SPLINE
SPL {X  -162.820, Y  +495.897, Z    +0.000, E1   +21.662, E3 +486078.194}
SPL {X  -162.820, Y  +493.717, Z    +0.000, E1   +21.704, E3 +486089.301}
SPL {X  -162.820, Y  +491.396, Z    +0.000, E1   +21.707, E3 +486101.424}
SPL {X  -162.820, Y  +489.485, Z    +0.000, E1   +21.661, E3 +486111.772}
SPL {X  -162.820, Y  +487.723, Z    +0.000, E1   +21.665, E3 +486120.976}
SPL {X  -162.820, Y  +485.661, Z    +0.000, E1   +21.712, E3 +486131.419}
SPL {X  -162.820, Y  +482.775, Z    +0.000, E1   +21.716, E3 +486146.672}
SPL {X  -162.820, Y  +479.894, Z    +0.000, E1   +21.695, E3 +486161.748}
SPL {X  -162.820, Y  +477.685, Z    +0.000, E1   +21.656, E3 +486173.685}
SPL {X  -162.820, Y  +475.419, Z    +0.000, E1   +21.711, E3 +486185.038}
SPL {X  -162.820, Y  +473.301, Z    +0.000, E1   +21.712, E3 +486196.135}
SPL {X  -162.820, Y  +470.965, Z    +0.000, E1   +21.700, E3 +486208.480}
SPL {X  -162.820, Y  +469.036, Z    +0.000, E1   +21.695, E3 +486218.524}
SPL {X  -162.820, Y  +467.138, Z    +0.000, E1   +21.678, E3 +486228.695}
SPL {X  -162.820, Y  +465.011, Z    +0.000, E1   +21.692, E3 +486239.678}
SPL {X  -162.820, Y  +462.669, Z    +0.000, E1   +21.752, E3 +486251.459}
SPL {X  -162.820, Y  +460.725, Z    +0.000, E1   +21.689, E3 +486262.072}
SPL {X  -162.820, Y  +458.666, Z    +0.000, E1   +21.695, E3 +486272.883}
SPL {X  -162.820, Y  +456.431, Z    +0.000, E1   +21.708, E3 +486284.412}
SPL {X  -162.820, Y  +453.609, Z    +0.000, E1   +21.757, E3 +486298.946}
SPL {X  -162.820, Y  +450.610, Z    +0.000, E1   +21.698, E3 +486315.003}
SPL {X  -162.820, Y  +448.170, Z    +0.000, E1   +21.667, E3 +486328.024}
SPL {X  -162.820, Y  +446.246, Z    +0.000, E1   +21.696, E3 +486337.842}
SPL {X  -162.820, Y  +443.784, Z    +0.000, E1   +21.713, E3 +486350.628}
SPL {X  -162.820, Y  +441.754, Z    +0.000, E1   +21.708, E3 +486361.180}
SPL {X  -162.820, Y  +439.933, Z    +0.000, E1   +21.690, E3 +486370.944}
SPL {X  -162.820, Y  +437.628, Z    +0.000, E1   +21.678, E3 +486383.132}
SPL {X  -162.820, Y  +435.262, Z    +0.000, E1   +21.727, E3 +486395.067}
SPL {X  -162.820, Y  +433.510, Z    +0.000, E1   +21.692, E3 +486404.481}
SPL {X  -162.820, Y  +431.492, Z    +0.000, E1   +21.686, E3 +486415.177}
SPL {X  -162.820, Y  +429.074, Z    +0.000, E1   +21.710, E3 +486427.629}
SPL {X  -162.820, Y  +427.020, Z    +0.000, E1   +21.674, E3 +486438.630}
SPL {X  -162.820, Y  +424.525, Z    +0.000, E1   +21.712, E3 +486451.543}
SPL {X  -162.820, Y  +421.144, Z    +0.000, E1   +21.719, E3 +486469.210}
SPL {X  -162.820, Y  +418.116, Z    +0.000, E1   +21.761, E3 +486484.541}
SPL {X  -162.820, Y  +416.127, Z    +0.000, E1   +21.715, E3 +486495.247}
SPL {X  -162.820, Y  +414.361, Z    +0.000, E1   +21.613, E3 +486505.434}
SPL {X  -162.820, Y  +412.134, Z    +0.000, E1   +21.697, E3 +486516.378}
SPL {X  -162.820, Y  +409.248, Z    +0.000, E1   +21.741, E3 +486531.314}
SPL {X  -162.820, Y  +406.238, Z    +0.000, E1   +21.697, E3 +486547.282}
SPL {X  -162.820, Y  +404.001, Z    +0.000, E1   +21.723, E3 +486558.711}
SPL {X  -162.820, Y  +402.223, Z    +0.000, E1   +21.697, E3 +486568.196}
SPL {X  -162.820, Y  +400.348, Z    +0.000, E1   +21.713, E3 +486577.922}
SPL {X  -162.820, Y  +398.298, Z    +0.000, E1   +21.721, E3 +486588.538}
SPL {X  -162.820, Y  +396.371, Z    +0.000, E1   +21.713, E3 +486598.720}
SPL {X  -162.820, Y  +394.508, Z    +0.000, E1   +21.616, E3 +486609.275}
SPL {X  -162.820, Y  +392.435, Z    +0.000, E1   +21.681, E3 +486619.629}
SPL {X  -162.820, Y  +389.390, Z    +0.000, E1   +21.742, E3 +486635.235}
SPL {X  -162.820, Y  +386.818, Z    +0.000, E1   +21.679, E3 +486648.994}
SPL {X  -162.820, Y  +384.697, Z    +0.000, E1   +21.693, E3 +486660.064}
SPL {X  -162.820, Y  +382.288, Z    +0.000, E1   +21.742, E3 +486672.188}
SPL {X  -162.817, Y  +379.520, Z    +0.000, E1   +21.723, E3 +486687.025}
SPL {X  -162.776, Y  +376.710, Z    +0.000, E1   +21.698, E3 +486701.765}
SPL {X  -162.707, Y  +374.438, Z    +0.000, E1   +21.688, E3 +486713.768}
SPL {X  -162.607, Y  +372.171, Z    +0.000, E1   +21.692, E3 +486725.568}
SPL {X  -162.494, Y  +370.197, Z    +0.000, E1   +21.655, E3 +486736.194}
SPL {X  -162.349, Y  +368.131, Z    +0.000, E1   +21.624, E3 +486747.312}
SPL {X  -162.161, Y  +365.866, Z    +0.000, E1   +21.642, E3 +486758.998}
SPL {X  -161.651, Y  +361.024, Z    +0.000, E1   +22.970, E3 +486772.421}
SPL {X  -160.281, Y  +351.857, Z    +0.000, E1   +24.243, E3 +486807.760}
ENDSPLINE

SPLINE
SPL {X  -161.833, Y  +362.603, Z    +0.000, E1   +17.021, E3 +486822.456}
ENDSPLINE

SPLINE
SPL {X  -160.786, Y  +354.842, Z    +0.000, E1   +19.274, E3 +486854.611}
ENDSPLINE

SPLINE
SPL {X  -162.485, Y  +370.062, Z    +0.000, E1   +10.606, E3 +486860.990}
SPL {X  -162.818, Y  +379.636, Z    +0.000, E1    +5.115, E3 +486850.338}
SPL {X  -162.820, Y  +386.976, Z    +0.000, E1    +0.144, E3 +486849.437}
SPL {X  -162.820, Y  +391.982, Z    +0.000, E1    -3.443, E3 +486856.202}
SPL {X  -162.820, Y  +399.630, Z    +0.000, E1    -9.426, E3 +486858.710}
SPL {X  -162.820, Y  +408.127, Z    +0.000, E1   -18.417, E3 +486844.998}
SPL {X  -162.820, Y  +420.083, Z    +0.000, E1   -24.325, E3 +486865.474}
SPL {X  -162.820, Y  +428.527, Z    +0.000, E1   -26.988, E3 +486882.766}
SPL {X  -162.820, Y  +431.336, Z    +0.000, E1   -24.162, E3 +486912.976}
SPL {X  -162.820, Y  +432.048, Z    +0.000, E1   -22.832, E3 +486927.480}
SPL {X  -162.820, Y  +434.888, Z    +0.000, E1   -22.823, E3 +486941.429}
SPL {X  -162.820, Y  +436.834, Z    +0.000, E1   -22.779, E3 +486951.389}
SPL {X  -162.820, Y  +438.868, Z    +0.000, E1   -22.837, E3 +486961.043}
SPL {X  -162.820, Y  +441.351, Z    +0.000, E1   -22.805, E3 +486973.618}
SPL {X  -162.820, Y  +443.809, Z    +0.000, E1   -22.804, E3 +486985.784}
SPL {X  -162.820, Y  +447.077, Z    +0.000, E1   -22.869, E3 +487001.595}
SPL {X  -162.820, Y  +449.911, Z    +0.000, E1   -22.774, E3 +487016.204}
SPL {X  -162.820, Y  +451.861, Z    +0.000, E1   -22.750, E3 +487026.052}
SPL {X  -162.820, Y  +454.167, Z    +0.000, E1   -22.842, E3 +487036.781}
SPL {X  -162.820, Y  +456.529, Z    +0.000, E1   -22.855, E3 +487048.310}
SPL {X  -162.820, Y  +458.725, Z    +0.000, E1   -22.793, E3 +487059.714}
SPL {X  -162.820, Y  +461.700, Z    +0.000, E1   -22.822, E3 +487074.336}
SPL {X  -162.820, Y  +464.633, Z    +0.000, E1   -22.813, E3 +487088.833}
SPL {X  -162.820, Y  +466.699, Z    +0.000, E1   -22.824, E3 +487098.879}
SPL {X  -162.820, Y  +468.655, Z    +0.000, E1   -22.858, E3 +487108.323}
SPL {X  -162.820, Y  +470.892, Z    +0.000, E1   -22.837, E3 +487119.562}
SPL {X  -162.820, Y  +473.485, Z    +0.000, E1   -22.806, E3 +487132.760}
SPL {X  -162.820, Y  +475.738, Z    +0.000, E1   -22.728, E3 +487144.425}
SPL {X  -162.820, Y  +478.177, Z    +0.000, E1   -22.834, E3 +487155.765}
SPL {X  -162.820, Y  +481.034, Z    +0.000, E1   -22.831, E3 +487169.902}
SPL {X  -162.820, Y  +483.391, Z    +0.000, E1   -22.793, E3 +487181.838}
SPL {X  -162.820, Y  +486.307, Z    +0.000, E1   -22.833, E3 +487196.092}
SPL {X  -162.820, Y  +489.750, Z    +0.000, E1   -22.832, E3 +487213.162}
SPL {X  -162.820, Y  +492.546, Z    +0.000, E1   -22.823, E3 +487226.920}
SPL {X  -162.820, Y  +495.526, Z    +0.000, E1   -22.833, E3 +487241.803}
SPL {X  -162.820, Y  +499.330, Z    +0.000, E1   -22.841, E3 +487260.584}
SPL {X  -162.820, Y  +502.361, Z    +0.000, E1   -22.801, E3 +487275.743}
SPL {X  -162.820, Y  +505.323, Z    +0.000, E1   -22.838, E3 +487290.215}
SPL {X  -162.820, Y  +508.611, Z    +0.000, E1   -22.838, E3 +487306.477}
SPL {X  -162.820, Y  +511.620, Z    +0.000, E1   -22.791, E3 +487321.721}
SPL {X  -162.820, Y  +513.873, Z    +0.000, E1   -22.800, E3 +487332.693}
SPL {X  -162.820, Y  +516.100, Z    +0.000, E1   -22.809, E3 +487343.770}
SPL {X  -162.820, Y  +518.662, Z    +0.000, E1   -22.847, E3 +487356.068}
SPL {X  -162.820, Y  +520.641, Z    +0.000, E1   -22.790, E3 +487366.309}
SPL {X  -162.820, Y  +522.740, Z    +0.000, E1   -22.811, E3 +487376.552}
SPL {X  -162.820, Y  +524.628, Z    +0.000, E1   -22.846, E3 +487385.547}
SPL {X  -162.820, Y  +526.661, Z    +0.000, E1   -22.801, E3 +487396.102}
SPL {X  -162.820, Y  +529.662, Z    +0.000, E1   -22.810, E3 +487410.953}
SPL {X  -162.820, Y  +532.614, Z    +0.000, E1   -22.828, E3 +487425.359}
SPL {X  -162.820, Y  +534.838, Z    +0.000, E1   -22.864, E3 +487435.988}
SPL {X  -162.820, Y  +536.882, Z    +0.000, E1   -22.782, E3 +487446.843}
SPL {X  -162.820, Y  +539.194, Z    +0.000, E1   -22.826, E3 +487457.891}
SPL {X  -162.820, Y  +541.555, Z    +0.000, E1   -22.817, E3 +487469.706}
SPL {X  -162.820, Y  +543.728, Z    +0.000, E1   -22.799, E3 +487480.563}
SPL {X  -162.820, Y  +545.925, Z    +0.000, E1   -22.803, E3 +487491.433}
SPL {X  -162.820, Y  +548.328, Z    +0.000, E1   -22.796, E3 +487503.429}
SPL {X  -162.820, Y  +551.027, Z    +0.000, E1   -22.819, E3 +487516.622}
SPL {X  -162.820, Y  +553.721, Z    +0.000, E1   -22.807, E3 +487530.066}
SPL {X  -162.820, Y  +556.430, Z    +0.000, E1   -22.821, E3 +487543.362}
SPL {X  -162.820, Y  +559.675, Z    +0.000, E1   -22.837, E3 +487559.442}
SPL {X  -162.820, Y  +562.799, Z    +0.000, E1   -22.814, E3 +487574.948}
SPL {X  -162.820, Y  +565.170, Z    +0.000, E1   -22.801, E3 +487586.773}
SPL {X  -162.820, Y  +568.020, Z    +0.000, E1   -22.787, E3 +487601.160}
SPL {X  -162.820, Y  +570.992, Z    +0.000, E1   -22.834, E3 +487615.379}
SPL {X  -162.820, Y  +572.901, Z    +0.000, E1   -22.775, E3 +487625.247}
SPL {X  -162.820, Y  +575.638, Z    +0.000, E1   -22.855, E3 +487638.357}
SPL {X  -162.820, Y  +578.553, Z    +0.000, E1   -22.801, E3 +487653.069}
SPL {X  -162.820, Y  +581.064, Z    +0.000, E1   -22.823, E3 +487665.354}
SPL {X  -162.820, Y  +583.435, Z    +0.000, E1   -22.808, E3 +487677.175}
SPL {X  -162.820, Y  +585.410, Z    +0.000, E1   -22.764, E3 +487687.311}
SPL {X  -162.820, Y  +587.676, Z    +0.000, E1   -22.853, E3 +487697.826}
SPL {X  -162.820, Y  +589.682, Z    +0.000, E1   -22.776, E3 +487708.355}
SPL {X  -162.820, Y  +591.720, Z    +0.000, E1   -22.868, E3 +487717.666}
SPL {X  -162.820, Y  +593.650, Z    +0.000, E1   -22.810, E3 +487727.736}
SPL {X  -162.820, Y  +595.830, Z    +0.000, E1   -22.828, E3 +487738.352}
SPL {X  -162.820, Y  +598.094, Z    +0.000, E1   -22.843, E3 +487749.465}
SPL {X  -162.820, Y  +600.420, Z    +0.000, E1   -22.826, E3 +487761.096}
SPL {X  -162.820, Y  +602.573, Z    +0.000, E1   -22.830, E3 +487771.682}
SPL {X  -162.820, Y  +604.828, Z    +0.000, E1   -22.784, E3 +487783.320}
SPL {X  -162.820, Y  +607.142, Z    +0.000, E1   -22.808, E3 +487794.501}
SPL {X  -162.820, Y  +608.890, Z    +0.000, E1   -22.790, E3 +487803.325}
SPL {X  -162.820, Y  +611.103, Z    +0.000, E1   -22.785, E3 +487814.363}
SPL {X  -162.820, Y  +613.294, Z    +0.000, E1   -22.780, E3 +487825.237}
SPL {X  -162.820, Y  +615.356, Z    +0.000, E1   -22.799, E3 +487835.294}
SPL {X  -162.820, Y  +617.439, Z    +0.000, E1   -22.808, E3 +487845.552}
SPL {X  -162.820, Y  +619.665, Z    +0.000, E1   -22.817, E3 +487856.520}
SPL {X  -162.820, Y  +621.733, Z    +0.000, E1   -22.759, E3 +487867.244}
SPL {X  -162.820, Y  +624.076, Z    +0.000, E1   -22.774, E3 +487878.749}
SPL {X  -162.820, Y  +626.527, Z    +0.000, E1   -22.768, E3 +487890.992}
SPL {X  -162.820, Y  +629.758, Z    +0.000, E1   -22.800, E3 +487906.921}
SPL {X  -162.820, Y  +632.572, Z    +0.000, E1   -22.785, E3 +487920.770}
SPL {X  -162.820, Y  +634.507, Z    +0.000, E1   -22.784, E3 +487930.409}
SPL {X  -162.820, Y  +636.863, Z    +0.000, E1   -22.760, E3 +487942.331}
SPL {X  -162.820, Y  +640.111, Z    +0.000, E1   -22.809, E3 +487958.214}
SPL {X  -162.820, Y  +643.449, Z    +0.000, E1   -22.796, E3 +487974.731}
SPL {X  -162.820, Y  +645.630, Z    +0.000, E1   -22.795, E3 +487985.428}
SPL {X  -162.820, Y  +647.561, Z    +0.000, E1   -22.705, E3 +487995.878}
SPL {X  -162.820, Y  +649.758, Z    +0.000, E1   -22.780, E3 +488006.068}
SPL {X  -162.820, Y  +651.708, Z    +0.000, E1   -22.810, E3 +488015.563}
SPL {X  -162.820, Y  +653.898, Z    +0.000, E1   -22.796, E3 +488026.484}
SPL {X  -162.820, Y  +656.161, Z    +0.000, E1   -22.812, E3 +488037.605}
SPL {X  -162.820, Y  +658.384, Z    +0.000, E1   -22.822, E3 +488048.471}
SPL {X  -162.820, Y  +660.215, Z    +0.000, E1   -22.649, E3 +488059.062}
SPL {X  -162.820, Y  +662.823, Z    +0.000, E1   -22.799, E3 +488070.770}
SPL {X  -162.820, Y  +665.112, Z    +0.000, E1   -22.835, E3 +488081.824}
SPL {X  -162.820, Y  +667.016, Z    +0.000, E1   -22.823, E3 +488091.253}
SPL {X  -162.820, Y  +668.960, Z    +0.000, E1   -22.773, E3 +488101.420}
SPL {X  -162.820, Y  +672.333, Z    +0.000, E1   -22.837, E3 +488117.756}
SPL {X  -162.812, Y  +675.071, Z    +0.000, E1   -22.742, E3 +488131.901}
SPL {X  -162.773, Y  +677.428, Z    +0.000, E1   -22.762, E3 +488143.499}
SPL {X  -162.691, Y  +679.987, Z    +0.000, E1   -22.794, E3 +488155.912}
SPL {X  -162.604, Y  +681.880, Z    +0.000, E1   -22.691, E3 +488166.073}
SPL {X  -162.458, Y  +684.346, Z    +0.000, E1   -22.764, E3 +488177.866}
SPL {X  -162.296, Y  +686.547, Z    +0.000, E1   -22.660, E3 +488189.483}
SPL {X  -162.090, Y  +688.902, Z    +0.000, E1   -22.700, E3 +488200.991}
SPL {X  -161.474, Y  +694.390, Z    +0.000, E1   -24.298, E3 +488214.347}
SPL {X  -158.730, Y  +709.763, Z    +0.000, E1   -31.225, E3 +488225.685}
ENDSPLINE

SPLINE
SPL {X  -160.932, Y  +698.225, Z    +0.000, E1   -21.712, E3 +488256.795}
SPL {X  -161.917, Y  +690.622, Z    +0.000, E1   -16.445, E3 +488270.395}
ENDSPLINE

SPLINE
SPL {X  -161.349, Y  +695.340, Z    +0.000, E1   -18.625, E3 +488278.014}
ENDSPLINE

SPLINE
SPL {X  -162.534, Y  +683.153, Z    +0.000, E1   -10.475, E3 +488299.144}
SPL {X  -162.820, Y  +667.630, Z    +0.000, E1    -0.882, E3 +488293.121}
SPL {X  -162.820, Y  +661.883, Z    +0.000, E1    +3.373, E3 +488298.564}
SPL {X  -162.820, Y  +653.808, Z    +0.000, E1    +9.891, E3 +488296.255}
SPL {X  -162.820, Y  +632.548, Z    +0.000, E1   +27.446, E3 +488292.792}
ENDSPLINE

SPLINE
SPL {X  -162.820, Y  +638.080, Z    +0.000, E1   +18.858, E3 +488320.540}
ENDSPLINE

SPLINE
SPL {X  -162.820, Y  +623.278, Z    +0.000, E1   +28.723, E3 +488322.111}
SPL {X  -162.820, Y  +618.658, Z    +0.000, E1   +26.841, E3 +488350.720}
ENDSPLINE

SPLINE
SPL {X  -162.820, Y  +623.685, Z    +0.000, E1   +22.346, E3 +488363.027}
ENDSPLINE

SPLINE
SPL {X  -162.820, Y  +621.304, Z    +0.000, E1   +22.259, E3 +488375.842}
SPL {X  -162.820, Y  +618.758, Z    +0.000, E1   +22.239, E3 +488388.993}
SPL {X  -162.820, Y  +616.062, Z    +0.000, E1   +22.275, E3 +488402.413}
SPL {X  -162.820, Y  +613.536, Z    +0.000, E1   +22.242, E3 +488415.535}
SPL {X  -162.820, Y  +610.461, Z    +0.000, E1   +22.264, E3 +488431.166}
SPL {X  -162.820, Y  +607.796, Z    +0.000, E1   +22.261, E3 +488444.537}
SPL {X  -162.820, Y  +605.178, Z    +0.000, E1   +22.267, E3 +488458.021}
SPL {X  -162.820, Y  +602.350, Z    +0.000, E1   +22.224, E3 +488472.638}
SPL {X  -162.820, Y  +599.842, Z    +0.000, E1   +22.298, E3 +488484.790}
SPL {X  -162.820, Y  +597.194, Z    +0.000, E1   +22.253, E3 +488498.711}
SPL {X  -162.820, Y  +594.779, Z    +0.000, E1   +22.284, E3 +488510.615}
SPL {X  -162.820, Y  +592.389, Z    +0.000, E1   +22.245, E3 +488523.231}
SPL {X  -162.820, Y  +589.492, Z    +0.000, E1   +22.304, E3 +488537.415}
SPL {X  -162.820, Y  +587.447, Z    +0.000, E1   +22.279, E3 +488547.944}
SPL {X  -162.820, Y  +585.192, Z    +0.000, E1   +22.298, E3 +488559.355}
SPL {X  -162.820, Y  +582.610, Z    +0.000, E1   +22.234, E3 +488572.978}
SPL {X  -162.820, Y  +580.317, Z    +0.000, E1   +22.300, E3 +488584.032}
SPL {X  -162.820, Y  +578.878, Z    +0.000, E1   +22.272, E3 +488591.541}
SPL {X  -162.820, Y  +576.856, Z    +0.000, E1   +22.233, E3 +488602.300}
SPL {X  -162.820, Y  +574.811, Z    +0.000, E1   +22.236, E3 +488612.563}
SPL {X  -162.820, Y  +572.645, Z    +0.000, E1   +22.246, E3 +488623.659}
SPL {X  -162.820, Y  +570.282, Z    +0.000, E1   +22.231, E3 +488635.709}
SPL {X  -162.820, Y  +567.961, Z    +0.000, E1   +22.247, E3 +488647.499}
SPL {X  -162.820, Y  +564.506, Z    +0.000, E1   +22.298, E3 +488664.813}
SPL {X  -162.820, Y  +561.620, Z    +0.000, E1   +22.191, E3 +488680.194}
SPL {X  -162.820, Y  +559.515, Z    +0.000, E1   +22.273, E3 +488690.196}
SPL {X  -162.820, Y  +556.723, Z    +0.000, E1   +22.309, E3 +488704.279}
SPL {X  -162.820, Y  +554.378, Z    +0.000, E1   +22.288, E3 +488716.125}
SPL {X  -162.820, Y  +552.787, Z    +0.000, E1   +22.213, E3 +488724.947}
SPL {X  -162.820, Y  +550.871, Z    +0.000, E1   +22.229, E3 +488734.541}
SPL {X  -162.820, Y  +548.168, Z    +0.000, E1   +22.298, E3 +488747.877}
SPL {X  -162.820, Y  +545.860, Z    +0.000, E1   +22.216, E3 +488760.135}
SPL {X  -162.820, Y  +543.558, Z    +0.000, E1   +22.285, E3 +488771.365}
SPL {X  -162.820, Y  +541.633, Z    +0.000, E1   +22.257, E3 +488781.294}
SPL {X  -162.820, Y  +539.116, Z    +0.000, E1   +22.302, E3 +488793.904}
SPL {X  -162.820, Y  +535.523, Z    +0.000, E1   +22.266, E3 +488812.566}
SPL {X  -162.820, Y  +531.757, Z    +0.000, E1   +22.276, E3 +488831.620}
SPL {X  -162.820, Y  +527.980, Z    +0.000, E1   +22.326, E3 +488850.451}
SPL {X  -162.820, Y  +524.599, Z    +0.000, E1   +22.287, E3 +488867.849}
SPL {X  -162.820, Y  +522.011, Z    +0.000, E1   +22.282, E3 +488880.926}
SPL {X  -162.820, Y  +519.457, Z    +0.000, E1   +22.481, E3 +488892.215}
SPL {X  -162.820, Y  +506.285, Z    +0.000, E1   +28.538, E3 +488903.673}
SPL {X  -162.820, Y  +504.441, Z    +0.000, E1   +27.574, E3 +488918.015}
SPL {X  -162.820, Y  +502.813, Z    +0.000, E1   +26.013, E3 +488936.213}
SPL {X  -162.820, Y  +502.016, Z    +0.000, E1   +24.802, E3 +488948.555}
SPL {X  -162.820, Y  +501.060, Z    +0.000, E1   +24.081, E3 +488958.745}
SPL {X  -162.820, Y  +500.336, Z    +0.000, E1   +23.110, E3 +488969.885}
SPL {X  -162.820, Y  +499.240, Z    +0.000, E1   +22.316, E3 +488982.196}
SPL {X  -162.820, Y  +498.027, Z    +0.000, E1   +21.516, E3 +488995.103}
SPL {X  -162.820, Y  +495.897, Z    +0.000, E1   +21.662, E3 +489005.023}
SPL {X  -162.820, Y  +493.717, Z    +0.000, E1   +21.704, E3 +489016.130}
SPL {X  -162.820, Y  +491.396, Z    +0.000, E1   +21.707, E3 +489028.254}
SPL {X  -162.820, Y  +488.560, Z    +0.000, E1   +21.695, E3 +489043.363}
SPL {X  -162.820, Y  +485.661, Z    +0.000, E1   +21.712, E3 +489058.248}
SPL {X  -162.820, Y  +483.668, Z    +0.000, E1   +21.664, E3 +489069.076}
SPL {X  -162.820, Y  +481.739, Z    +0.000, E1   +21.704, E3 +489078.790}
SPL {X  -162.820, Y  +479.894, Z    +0.000, E1   +21.695, E3 +489088.577}
SPL {X  -162.820, Y  +477.685, Z    +0.000, E1   +21.656, E3 +489100.515}
SPL {X  -162.820, Y  +475.419, Z    +0.000, E1   +21.711, E3 +489111.867}
SPL {X  -162.820, Y  +473.301, Z    +0.000, E1   +21.712, E3 +489122.964}
SPL {X  -162.820, Y  +470.965, Z    +0.000, E1   +21.700, E3 +489135.309}
SPL {X  -162.820, Y  +469.036, Z    +0.000, E1   +21.695, E3 +489145.353}
SPL {X  -162.820, Y  +467.138, Z    +0.000, E1   +21.678, E3 +489155.525}
SPL {X  -162.820, Y  +465.011, Z    +0.000, E1   +21.692, E3 +489166.507}
SPL {X  -162.820, Y  +462.669, Z    +0.000, E1   +21.752, E3 +489178.288}
SPL {X  -162.820, Y  +460.725, Z    +0.000, E1   +21.689, E3 +489188.901}
SPL {X  -162.820, Y  +458.666, Z    +0.000, E1   +21.695, E3 +489199.713}
SPL {X  -162.820, Y  +456.431, Z    +0.000, E1   +21.708, E3 +489211.241}
SPL {X  -162.820, Y  +453.609, Z    +0.000, E1   +21.757, E3 +489225.775}
SPL {X  -162.820, Y  +450.610, Z    +0.000, E1   +21.698, E3 +489241.832}
SPL {X  -162.820, Y  +448.170, Z    +0.000, E1   +21.667, E3 +489254.853}
SPL {X  -162.820, Y  +446.246, Z    +0.000, E1   +21.696, E3 +489264.671}
SPL {X  -162.820, Y  +443.784, Z    +0.000, E1   +21.713, E3 +489277.457}
SPL {X  -162.820, Y  +440.567, Z    +0.000, E1   +21.731, E3 +489294.297}
SPL {X  -162.820, Y  +437.628, Z    +0.000, E1   +21.678, E3 +489309.961}
SPL {X  -162.820, Y  +434.473, Z    +0.000, E1   +21.747, E3 +489326.057}
SPL {X  -162.820, Y  +431.492, Z    +0.000, E1   +21.686, E3 +489342.006}
SPL {X  -162.820, Y  +429.074, Z    +0.000, E1   +21.710, E3 +489354.458}
SPL {X  -162.820, Y  +426.023, Z    +0.000, E1   +21.718, E3 +489370.526}
SPL {X  -162.820, Y  +422.986, Z    +0.000, E1   +21.685, E3 +489386.573}
SPL {X  -162.820, Y  +420.528, Z    +0.000, E1   +21.706, E3 +489399.223}
SPL {X  -162.820, Y  +418.116, Z    +0.000, E1   +21.761, E3 +489411.371}
SPL {X  -162.820, Y  +416.127, Z    +0.000, E1   +21.715, E3 +489422.076}
SPL {X  -162.820, Y  +414.361, Z    +0.000, E1   +21.613, E3 +489432.263}
SPL {X  -162.820, Y  +412.134, Z    +0.000, E1   +21.697, E3 +489443.208}
SPL {X  -162.820, Y  +409.248, Z    +0.000, E1   +21.741, E3 +489458.143}
SPL {X  -162.820, Y  +406.238, Z    +0.000, E1   +21.697, E3 +489474.111}
SPL {X  -162.820, Y  +404.001, Z    +0.000, E1   +21.723, E3 +489485.541}
SPL {X  -162.820, Y  +402.223, Z    +0.000, E1   +21.697, E3 +489495.026}
SPL {X  -162.820, Y  +400.348, Z    +0.000, E1   +21.713, E3 +489504.752}
SPL {X  -162.820, Y  +398.298, Z    +0.000, E1   +21.721, E3 +489515.367}
SPL {X  -162.820, Y  +396.371, Z    +0.000, E1   +21.713, E3 +489525.549}
SPL {X  -162.820, Y  +394.508, Z    +0.000, E1   +21.616, E3 +489536.104}
SPL {X  -162.820, Y  +392.435, Z    +0.000, E1   +21.681, E3 +489546.458}
SPL {X  -162.820, Y  +389.390, Z    +0.000, E1   +21.742, E3 +489562.065}
SPL {X  -162.820, Y  +386.818, Z    +0.000, E1   +21.679, E3 +489575.823}
SPL {X  -162.820, Y  +384.697, Z    +0.000, E1   +21.693, E3 +489586.894}
SPL {X  -162.820, Y  +382.288, Z    +0.000, E1   +21.742, E3 +489599.017}
SPL {X  -162.820, Y  +380.381, Z    +0.000, E1   +21.655, E3 +489609.742}
SPL {X  -162.808, Y  +378.512, Z    +0.000, E1   +21.736, E3 +489618.795}
SPL {X  -162.776, Y  +376.710, Z    +0.000, E1   +21.698, E3 +489628.594}
SPL {X  -162.707, Y  +374.438, Z    +0.000, E1   +21.688, E3 +489640.598}
SPL {X  -162.607, Y  +372.171, Z    +0.000, E1   +21.692, E3 +489652.397}
SPL {X  -162.494, Y  +370.197, Z    +0.000, E1   +21.655, E3 +489663.024}
SPL {X  -162.349, Y  +368.131, Z    +0.000, E1   +21.624, E3 +489674.142}
SPL {X  -162.161, Y  +365.866, Z    +0.000, E1   +21.642, E3 +489685.827}
SPL {X  -161.927, Y  +363.466, Z    +0.000, E1   +21.730, E3 +489697.598}
SPL {X  -160.290, Y  +351.907, Z    +0.000, E1   +27.562, E3 +489705.176}
SPL {X  -159.725, Y  +348.905, Z    +0.000, E1   +26.136, E3 +489730.411}
ENDSPLINE

SPLINE
SPL {X  -160.871, Y  +355.385, Z    +0.000, E1   +21.841, E3 +489739.254}
SPL {X  -161.833, Y  +362.603, Z    +0.000, E1   +17.021, E3 +489749.285}
ENDSPLINE

SPLINE
SPL {X  -160.786, Y  +354.842, Z    +0.000, E1   +19.274, E3 +489781.441}
ENDSPLINE

SPLINE
SPL {X  -162.485, Y  +370.062, Z    +0.000, E1   +10.606, E3 +489787.819}
SPL {X  -162.818, Y  +379.636, Z    +0.000, E1    +5.115, E3 +489777.168}
SPL {X  -162.820, Y  +386.976, Z    +0.000, E1    +0.144, E3 +489776.267}
SPL {X  -162.820, Y  +390.236, Z    +0.000, E1    -2.204, E3 +489782.325}
SPL {X  -162.820, Y  +393.415, Z    +0.000, E1    -4.587, E3 +489783.609}
SPL {X  -162.820, Y  +399.630, Z    +0.000, E1    -9.426, E3 +489785.539}
SPL {X  -162.820, Y  +408.127, Z    +0.000, E1   -18.417, E3 +489771.827}
SPL {X  -162.820, Y  +420.083, Z    +0.000, E1   -24.325, E3 +489792.303}
SPL {X  -162.820, Y  +428.527, Z    +0.000, E1   -26.988, E3 +489809.595}
SPL {X  -162.820, Y  +431.336, Z    +0.000, E1   -24.162, E3 +489839.805}
SPL {X  -162.820, Y  +432.048, Z    +0.000, E1   -22.832, E3 +489854.309}
SPL {X  -162.820, Y  +434.888, Z    +0.000, E1   -22.823, E3 +489868.258}
SPL {X  -162.820, Y  +436.834, Z    +0.000, E1   -22.779, E3 +489878.218}
SPL {X  -162.820, Y  +438.868, Z    +0.000, E1   -22.837, E3 +489887.872}
SPL {X  -162.820, Y  +441.351, Z    +0.000, E1   -22.805, E3 +489900.447}
SPL {X  -162.820, Y  +443.809, Z    +0.000, E1   -22.804, E3 +489912.613}
SPL {X  -162.820, Y  +447.077, Z    +0.000, E1   -22.869, E3 +489928.424}
SPL {X  -162.820, Y  +449.911, Z    +0.000, E1   -22.774, E3 +489943.033}
SPL {X  -162.820, Y  +451.861, Z    +0.000, E1   -22.750, E3 +489952.881}
SPL {X  -162.820, Y  +454.167, Z    +0.000, E1   -22.842, E3 +489963.610}
SPL {X  -162.820, Y  +456.529, Z    +0.000, E1   -22.855, E3 +489975.139}
SPL {X  -162.820, Y  +458.725, Z    +0.000, E1   -22.793, E3 +489986.543}
SPL {X  -162.820, Y  +460.754, Z    +0.000, E1   -22.806, E3 +489996.416}
SPL {X  -162.820, Y  +462.409, Z    +0.000, E1   -22.783, E3 +490004.833}
SPL {X  -162.820, Y  +464.633, Z    +0.000, E1   -22.813, E3 +490015.662}
SPL {X  -162.820, Y  +467.913, Z    +0.000, E1   -22.879, E3 +490031.501}
SPL {X  -162.820, Y  +470.892, Z    +0.000, E1   -22.837, E3 +490046.391}
SPL {X  -162.820, Y  +472.726, Z    +0.000, E1   -22.777, E3 +490055.930}
SPL {X  -162.820, Y  +475.118, Z    +0.000, E1   -22.777, E3 +490067.901}
SPL {X  -162.820, Y  +477.389, Z    +0.000, E1   -22.803, E3 +490078.818}
SPL {X  -162.820, Y  +478.914, Z    +0.000, E1   -22.821, E3 +490086.209}
SPL {X  -162.820, Y  +481.034, Z    +0.000, E1   -22.831, E3 +490096.731}
SPL {X  -162.820, Y  +484.256, Z    +0.000, E1   -22.840, E3 +490112.750}
SPL {X  -162.820, Y  +487.952, Z    +0.000, E1   -22.824, E3 +490131.180}
SPL {X  -162.820, Y  +491.768, Z    +0.000, E1   -22.852, E3 +490149.861}
SPL {X  -162.820, Y  +495.526, Z    +0.000, E1   -22.833, E3 +490168.632}
SPL {X  -162.820, Y  +499.330, Z    +0.000, E1   -22.841, E3 +490187.413}
SPL {X  -162.820, Y  +503.049, Z    +0.000, E1   -22.823, E3 +490205.963}
SPL {X  -162.820, Y  +506.908, Z    +0.000, E1   -22.877, E3 +490224.633}
SPL {X  -162.820, Y  +510.068, Z    +0.000, E1   -22.761, E3 +490241.104}
SPL {X  -162.820, Y  +512.359, Z    +0.000, E1   -22.823, E3 +490251.836}
SPL {X  -162.820, Y  +514.562, Z    +0.000, E1   -22.806, E3 +490263.023}
SPL {X  -162.820, Y  +517.952, Z    +0.000, E1   -22.864, E3 +490279.420}
SPL {X  -162.820, Y  +520.641, Z    +0.000, E1   -22.790, E3 +490293.139}
SPL {X  -162.820, Y  +522.740, Z    +0.000, E1   -22.811, E3 +490303.381}
SPL {X  -162.820, Y  +524.628, Z    +0.000, E1   -22.846, E3 +490312.376}
SPL {X  -162.820, Y  +526.661, Z    +0.000, E1   -22.801, E3 +490322.931}
SPL {X  -162.820, Y  +529.662, Z    +0.000, E1   -22.810, E3 +490337.782}
SPL {X  -162.820, Y  +532.614, Z    +0.000, E1   -22.828, E3 +490352.188}
SPL {X  -162.820, Y  +534.838, Z    +0.000, E1   -22.864, E3 +490362.817}
SPL {X  -162.820, Y  +536.882, Z    +0.000, E1   -22.782, E3 +490373.672}
SPL {X  -162.820, Y  +539.194, Z    +0.000, E1   -22.826, E3 +490384.721}
SPL {X  -162.820, Y  +541.555, Z    +0.000, E1   -22.817, E3 +490396.535}
SPL {X  -162.820, Y  +543.728, Z    +0.000, E1   -22.799, E3 +490407.393}
SPL {X  -162.820, Y  +545.925, Z    +0.000, E1   -22.803, E3 +490418.262}
SPL {X  -162.820, Y  +548.328, Z    +0.000, E1   -22.796, E3 +490430.258}
SPL {X  -162.820, Y  +551.027, Z    +0.000, E1   -22.819, E3 +490443.451}
SPL {X  -162.820, Y  +553.721, Z    +0.000, E1   -22.807, E3 +490456.895}
SPL {X  -162.820, Y  +556.430, Z    +0.000, E1   -22.821, E3 +490470.191}
SPL {X  -162.820, Y  +558.974, Z    +0.000, E1   -22.806, E3 +490482.891}
SPL {X  -162.820, Y  +562.171, Z    +0.000, E1   -22.845, E3 +490498.589}
SPL {X  -162.820, Y  +565.170, Z    +0.000, E1   -22.801, E3 +490513.602}
SPL {X  -162.820, Y  +567.308, Z    +0.000, E1   -22.750, E3 +490524.618}
SPL {X  -162.820, Y  +570.378, Z    +0.000, E1   -22.843, E3 +490539.242}
SPL {X  -162.820, Y  +573.634, Z    +0.000, E1   -22.827, E3 +490555.386}
SPL {X  -162.820, Y  +576.228, Z    +0.000, E1   -22.814, E3 +490568.282}
SPL {X  -162.820, Y  +578.553, Z    +0.000, E1   -22.801, E3 +490579.898}
SPL {X  -162.820, Y  +581.064, Z    +0.000, E1   -22.823, E3 +490592.183}
SPL {X  -162.820, Y  +583.435, Z    +0.000, E1   -22.808, E3 +490604.004}
SPL {X  -162.820, Y  +585.410, Z    +0.000, E1   -22.764, E3 +490614.140}
SPL {X  -162.820, Y  +587.676, Z    +0.000, E1   -22.853, E3 +490624.655}
SPL {X  -162.820, Y  +590.707, Z    +0.000, E1   -22.855, E3 +490639.805}
SPL {X  -162.820, Y  +593.650, Z    +0.000, E1   -22.810, E3 +490654.565}
SPL {X  -162.820, Y  +595.830, Z    +0.000, E1   -22.828, E3 +490665.181}
SPL {X  -162.820, Y  +598.094, Z    +0.000, E1   -22.843, E3 +490676.294}
SPL {X  -162.820, Y  +600.420, Z    +0.000, E1   -22.826, E3 +490687.926}
SPL {X  -162.820, Y  +602.573, Z    +0.000, E1   -22.830, E3 +490698.511}
SPL {X  -162.820, Y  +604.828, Z    +0.000, E1   -22.784, E3 +490710.149}
SPL {X  -162.820, Y  +607.142, Z    +0.000, E1   -22.808, E3 +490721.330}
SPL {X  -162.820, Y  +608.890, Z    +0.000, E1   -22.790, E3 +490730.154}
SPL {X  -162.820, Y  +611.103, Z    +0.000, E1   -22.785, E3 +490741.193}
SPL {X  -162.820, Y  +613.294, Z    +0.000, E1   -22.780, E3 +490752.066}
SPL {X  -162.820, Y  +615.356, Z    +0.000, E1   -22.799, E3 +490762.123}
SPL {X  -162.820, Y  +617.439, Z    +0.000, E1   -22.808, E3 +490772.381}
SPL {X  -162.820, Y  +619.665, Z    +0.000, E1   -22.817, E3 +490783.349}
SPL {X  -162.820, Y  +621.733, Z    +0.000, E1   -22.759, E3 +490794.073}
SPL {X  -162.820, Y  +624.076, Z    +0.000, E1   -22.774, E3 +490805.578}
SPL {X  -162.820, Y  +627.244, Z    +0.000, E1   -22.803, E3 +490821.261}
SPL {X  -162.820, Y  +630.349, Z    +0.000, E1   -22.766, E3 +490836.793}
SPL {X  -162.820, Y  +632.572, Z    +0.000, E1   -22.785, E3 +490847.599}
SPL {X  -162.820, Y  +634.507, Z    +0.000, E1   -22.784, E3 +490857.238}
SPL {X  -162.820, Y  +636.863, Z    +0.000, E1   -22.760, E3 +490869.160}
SPL {X  -162.820, Y  +640.111, Z    +0.000, E1   -22.809, E3 +490885.043}
SPL {X  -162.820, Y  +643.449, Z    +0.000, E1   -22.796, E3 +490901.561}
SPL {X  -162.820, Y  +645.630, Z    +0.000, E1   -22.795, E3 +490912.257}
SPL {X  -162.820, Y  +647.561, Z    +0.000, E1   -22.705, E3 +490922.707}
SPL {X  -162.820, Y  +651.051, Z    +0.000, E1   -22.833, E3 +490939.127}
SPL {X  -162.820, Y  +653.898, Z    +0.000, E1   -22.796, E3 +490953.313}
SPL {X  -162.820, Y  +656.161, Z    +0.000, E1   -22.812, E3 +490964.434}
SPL {X  -162.820, Y  +658.384, Z    +0.000, E1   -22.822, E3 +490975.301}
SPL {X  -162.820, Y  +660.215, Z    +0.000, E1   -22.649, E3 +490985.891}
SPL {X  -162.820, Y  +662.823, Z    +0.000, E1   -22.799, E3 +490997.599}
SPL {X  -162.820, Y  +665.112, Z    +0.000, E1   -22.835, E3 +491008.654}
SPL {X  -162.820, Y  +667.016, Z    +0.000, E1   -22.823, E3 +491018.082}
SPL {X  -162.820, Y  +668.960, Z    +0.000, E1   -22.773, E3 +491028.249}
SPL {X  -162.820, Y  +671.605, Z    +0.000, E1   -22.777, E3 +491041.323}
SPL {X  -162.817, Y  +674.515, Z    +0.000, E1   -22.816, E3 +491055.520}
SPL {X  -162.773, Y  +677.428, Z    +0.000, E1   -22.762, E3 +491070.328}
SPL {X  -162.691, Y  +679.987, Z    +0.000, E1   -22.794, E3 +491082.741}
SPL {X  -162.559, Y  +682.717, Z    +0.000, E1   -22.726, E3 +491096.925}
SPL {X  -162.349, Y  +685.880, Z    +0.000, E1   -22.738, E3 +491112.526}
SPL {X  -162.090, Y  +688.902, Z    +0.000, E1   -22.700, E3 +491127.821}
SPL {X  -161.474, Y  +694.390, Z    +0.000, E1   -24.298, E3 +491141.176}
SPL {X  -158.553, Y  +710.529, Z    +0.000, E1   -30.890, E3 +491157.738}
ENDSPLINE

SPLINE
SPL {X  -161.215, Y  +696.305, Z    +0.000, E1   -20.575, E3 +491184.318}
SPL {X  -161.691, Y  +692.643, Z    +0.000, E1   -17.369, E3 +491200.507}
SPL {X  -162.534, Y  +683.153, Z    +0.000, E1   -10.475, E3 +491225.974}
SPL {X  -162.820, Y  +667.630, Z    +0.000, E1    -0.882, E3 +491219.950}
SPL {X  -162.820, Y  +661.883, Z    +0.000, E1    +3.373, E3 +491225.393}
SPL {X  -162.820, Y  +653.808, Z    +0.000, E1    +9.891, E3 +491223.085}
SPL {X  -162.820, Y  +632.548, Z    +0.000, E1   +27.446, E3 +491219.621}
ENDSPLINE

SPLINE
SPL {X  -162.820, Y  +638.080, Z    +0.000, E1   +18.858, E3 +491247.370}
ENDSPLINE

SPLINE
SPL {X  -162.820, Y  +623.278, Z    +0.000, E1   +28.723, E3 +491248.940}
SPL {X  -162.820, Y  +618.658, Z    +0.000, E1   +26.841, E3 +491277.549}
ENDSPLINE

SPLINE
SPL {X  -162.820, Y  +623.685, Z    +0.000, E1   +22.346, E3 +491289.856}
ENDSPLINE

SPLINE
SPL {X  -162.820, Y  +621.304, Z    +0.000, E1   +22.259, E3 +491302.671}
SPL {X  -162.820, Y  +618.758, Z    +0.000, E1   +22.239, E3 +491315.822}
SPL {X  -162.820, Y  +616.062, Z    +0.000, E1   +22.275, E3 +491329.242}
SPL {X  -162.820, Y  +613.536, Z    +0.000, E1   +22.242, E3 +491342.364}
SPL {X  -162.820, Y  +611.128, Z    +0.000, E1   +22.252, E3 +491354.535}
SPL {X  -162.820, Y  +608.428, Z    +0.000, E1   +22.255, E3 +491368.318}
SPL {X  -162.820, Y  +605.984, Z    +0.000, E1   +22.221, E3 +491380.955}
SPL {X  -162.820, Y  +603.020, Z    +0.000, E1   +22.272, E3 +491395.853}
SPL {X  -162.820, Y  +599.168, Z    +0.000, E1   +22.310, E3 +491415.121}
SPL {X  -162.820, Y  +596.569, Z    +0.000, E1   +22.222, E3 +491428.844}
SPL {X  -162.820, Y  +594.115, Z    +0.000, E1   +22.273, E3 +491441.069}
SPL {X  -162.820, Y  +591.721, Z    +0.000, E1   +22.239, E3 +491453.384}
SPL {X  -162.820, Y  +589.492, Z    +0.000, E1   +22.304, E3 +491464.245}
SPL {X  -162.820, Y  +587.447, Z    +0.000, E1   +22.279, E3 +491474.774}
SPL {X  -162.820, Y  +585.192, Z    +0.000, E1   +22.298, E3 +491486.184}
SPL {X  -162.820, Y  +582.610, Z    +0.000, E1   +22.234, E3 +491499.807}
SPL {X  -162.820, Y  +580.317, Z    +0.000, E1   +22.300, E3 +491510.861}
SPL {X  -162.820, Y  +578.878, Z    +0.000, E1   +22.272, E3 +491518.371}
SPL {X  -162.820, Y  +576.856, Z    +0.000, E1   +22.233, E3 +491529.129}
SPL {X  -162.820, Y  +573.830, Z    +0.000, E1   +22.272, E3 +491544.265}
SPL {X  -162.820, Y  +570.852, Z    +0.000, E1   +22.234, E3 +491559.725}
SPL {X  -162.820, Y  +568.608, Z    +0.000, E1   +22.253, E3 +491570.858}
SPL {X  -162.820, Y  +565.838, Z    +0.000, E1   +22.271, E3 +491585.089}
SPL {X  -162.820, Y  +562.162, Z    +0.000, E1   +22.252, E3 +491603.906}
SPL {X  -162.820, Y  +558.919, Z    +0.000, E1   +22.286, E3 +491620.070}
SPL {X  -162.820, Y  +555.548, Z    +0.000, E1   +22.322, E3 +491636.979}
SPL {X  -162.820, Y  +552.787, Z    +0.000, E1   +22.213, E3 +491651.776}
SPL {X  -162.820, Y  +550.136, Z    +0.000, E1   +22.258, E3 +491665.010}
SPL {X  -162.820, Y  +546.694, Z    +0.000, E1   +22.290, E3 +491682.332}
SPL {X  -162.820, Y  +543.558, Z    +0.000, E1   +22.285, E3 +491698.195}
SPL {X  -162.820, Y  +541.633, Z    +0.000, E1   +22.257, E3 +491708.123}
SPL {X  -162.820, Y  +539.116, Z    +0.000, E1   +22.302, E3 +491720.733}
SPL {X  -162.820, Y  +536.913, Z    +0.000, E1   +22.192, E3 +491732.658}
SPL {X  -162.820, Y  +534.880, Z    +0.000, E1   +22.252, E3 +491742.611}
SPL {X  -162.820, Y  +532.896, Z    +0.000, E1   +22.234, E3 +491752.772}
SPL {X  -162.820, Y  +531.056, Z    +0.000, E1   +22.251, E3 +491762.054}
SPL {X  -162.820, Y  +528.708, Z    +0.000, E1   +22.319, E3 +491773.435}
SPL {X  -162.820, Y  +525.932, Z    +0.000, E1   +22.258, E3 +491788.192}
SPL {X  -162.820, Y  +522.524, Z    +0.000, E1   +22.326, E3 +491804.916}
SPL {X  -162.820, Y  +519.457, Z    +0.000, E1   +22.481, E3 +491819.044}
SPL {X  -162.820, Y  +506.285, Z    +0.000, E1   +28.538, E3 +491830.502}
SPL {X  -162.820, Y  +504.441, Z    +0.000, E1   +27.574, E3 +491844.845}
SPL {X  -162.820, Y  +502.813, Z    +0.000, E1   +26.013, E3 +491863.042}
SPL {X  -162.820, Y  +502.016, Z    +0.000, E1   +24.802, E3 +491875.385}
SPL {X  -162.820, Y  +501.060, Z    +0.000, E1   +24.081, E3 +491885.574}
SPL {X  -162.820, Y  +499.934, Z    +0.000, E1   +22.814, E3 +491901.443}
SPL {X  -162.820, Y  +498.303, Z    +0.000, E1   +21.749, E3 +491918.699}
SPL {X  -162.820, Y  +495.897, Z    +0.000, E1   +21.662, E3 +491931.853}
SPL {X  -162.820, Y  +493.717, Z    +0.000, E1   +21.704, E3 +491942.959}
SPL {X  -162.820, Y  +491.396, Z    +0.000, E1   +21.707, E3 +491955.083}
SPL {X  -162.820, Y  +489.485, Z    +0.000, E1   +21.661, E3 +491965.431}
SPL {X  -162.820, Y  +487.723, Z    +0.000, E1   +21.665, E3 +491974.634}
SPL {X  -162.820, Y  +485.661, Z    +0.000, E1   +21.712, E3 +491985.078}
SPL {X  -162.820, Y  +482.775, Z    +0.000, E1   +21.716, E3 +492000.330}
SPL {X  -162.820, Y  +479.894, Z    +0.000, E1   +21.695, E3 +492015.406}
SPL {X  -162.820, Y  +477.685, Z    +0.000, E1   +21.656, E3 +492027.344}
SPL {X  -162.820, Y  +475.419, Z    +0.000, E1   +21.711, E3 +492038.697}
SPL {X  -162.820, Y  +473.301, Z    +0.000, E1   +21.712, E3 +492049.794}
SPL {X  -162.820, Y  +470.965, Z    +0.000, E1   +21.700, E3 +492062.139}
SPL {X  -162.820, Y  +469.036, Z    +0.000, E1   +21.695, E3 +492072.182}
SPL {X  -162.820, Y  +467.138, Z    +0.000, E1   +21.678, E3 +492082.354}
SPL {X  -162.820, Y  +465.011, Z    +0.000, E1   +21.692, E3 +492093.337}
SPL {X  -162.820, Y  +462.669, Z    +0.000, E1   +21.752, E3 +492105.117}
SPL {X  -162.820, Y  +460.725, Z    +0.000, E1   +21.689, E3 +492115.730}
SPL {X  -162.820, Y  +458.666, Z    +0.000, E1   +21.695, E3 +492126.542}
SPL {X  -162.820, Y  +456.431, Z    +0.000, E1   +21.708, E3 +492138.071}
SPL {X  -162.820, Y  +454.628, Z    +0.000, E1   +21.674, E3 +492147.789}
SPL {X  -162.820, Y  +452.690, Z    +0.000, E1   +21.773, E3 +492157.063}
SPL {X  -162.820, Y  +450.610, Z    +0.000, E1   +21.698, E3 +492168.662}
SPL {X  -162.820, Y  +448.170, Z    +0.000, E1   +21.667, E3 +492181.683}
SPL {X  -162.820, Y  +445.508, Z    +0.000, E1   +21.732, E3 +492195.201}
SPL {X  -162.820, Y  +442.443, Z    +0.000, E1   +21.712, E3 +492211.321}
SPL {X  -162.820, Y  +439.933, Z    +0.000, E1   +21.690, E3 +492224.602}
SPL {X  -162.820, Y  +437.628, Z    +0.000, E1   +21.678, E3 +492236.790}
SPL {X  -162.820, Y  +434.473, Z    +0.000, E1   +21.747, E3 +492252.887}
SPL {X  -162.820, Y  +431.492, Z    +0.000, E1   +21.686, E3 +492268.835}
SPL {X  -162.820, Y  +429.074, Z    +0.000, E1   +21.710, E3 +492281.287}
SPL {X  -162.820, Y  +426.023, Z    +0.000, E1   +21.718, E3 +492297.355}
SPL {X  -162.820, Y  +422.986, Z    +0.000, E1   +21.685, E3 +492313.403}
SPL {X  -162.820, Y  +420.528, Z    +0.000, E1   +21.706, E3 +492326.053}
SPL {X  -162.820, Y  +418.116, Z    +0.000, E1   +21.761, E3 +492338.200}
SPL {X  -162.820, Y  +416.127, Z    +0.000, E1   +21.715, E3 +492348.905}
SPL {X  -162.820, Y  +414.361, Z    +0.000, E1   +21.613, E3 +492359.092}
SPL {X  -162.820, Y  +411.450, Z    +0.000, E1   +21.710, E3 +492373.666}
SPL {X  -162.820, Y  +408.590, Z    +0.000, E1   +21.735, E3 +492388.291}
SPL {X  -162.820, Y  +406.238, Z    +0.000, E1   +21.697, E3 +492400.940}
SPL {X  -162.820, Y  +403.166, Z    +0.000, E1   +21.746, E3 +492416.746}
SPL {X  -162.820, Y  +400.348, Z    +0.000, E1   +21.713, E3 +492431.581}
SPL {X  -162.820, Y  +398.298, Z    +0.000, E1   +21.721, E3 +492442.196}
SPL {X  -162.820, Y  +396.371, Z    +0.000, E1   +21.713, E3 +492452.378}
SPL {X  -162.820, Y  +394.508, Z    +0.000, E1   +21.616, E3 +492462.934}
SPL {X  -162.820, Y  +391.777, Z    +0.000, E1   +21.714, E3 +492476.593}
SPL {X  -162.820, Y  +388.822, Z    +0.000, E1   +21.717, E3 +492491.913}
SPL {X  -162.820, Y  +386.818, Z    +0.000, E1   +21.679, E3 +492502.653}
SPL {X  -162.820, Y  +384.697, Z    +0.000, E1   +21.693, E3 +492513.723}
SPL {X  -162.820, Y  +382.288, Z    +0.000, E1   +21.742, E3 +492525.846}
SPL {X  -162.817, Y  +379.520, Z    +0.000, E1   +21.723, E3 +492540.684}
SPL {X  -162.776, Y  +376.710, Z    +0.000, E1   +21.698, E3 +492555.423}
SPL {X  -162.707, Y  +374.438, Z    +0.000, E1   +21.688, E3 +492567.427}
SPL {X  -162.607, Y  +372.171, Z    +0.000, E1   +21.692, E3 +492579.227}
SPL {X  -162.494, Y  +370.197, Z    +0.000, E1   +21.655, E3 +492589.853}
SPL {X  -162.349, Y  +368.131, Z    +0.000, E1   +21.624, E3 +492600.971}
SPL {X  -162.161, Y  +365.866, Z    +0.000, E1   +21.642, E3 +492612.656}
SPL {X  -161.651, Y  +361.024, Z    +0.000, E1   +22.970, E3 +492626.079}
SPL {X  -160.281, Y  +351.857, Z    +0.000, E1   +24.243, E3 +492661.418}
ENDSPLINE

SPLINE
SPL {X  -161.833, Y  +362.603, Z    +0.000, E1   +17.021, E3 +492676.114}
ENDSPLINE

SPLINE
SPL {X  -160.786, Y  +354.842, Z    +0.000, E1   +19.274, E3 +492708.270}
ENDSPLINE

SPLINE
SPL {X  -162.485, Y  +370.062, Z    +0.000, E1   +10.606, E3 +492714.648}
SPL {X  -162.818, Y  +379.636, Z    +0.000, E1    +5.115, E3 +492703.997}
SPL {X  -162.820, Y  +386.976, Z    +0.000, E1    +0.144, E3 +492703.096}
SPL {X  -162.820, Y  +390.236, Z    +0.000, E1    -2.204, E3 +492709.155}
SPL {X  -162.820, Y  +393.415, Z    +0.000, E1    -4.587, E3 +492710.439}
SPL {X  -162.820, Y  +399.630, Z    +0.000, E1    -9.426, E3 +492712.368}
SPL {X  -162.820, Y  +408.127, Z    +0.000, E1   -18.417, E3 +492698.657}
SPL {X  -162.820, Y  +420.083, Z    +0.000, E1   -24.325, E3 +492719.132}
SPL {X  -162.820, Y  +428.527, Z    +0.000, E1   -26.988, E3 +492736.424}
SPL {X  -162.820, Y  +431.191, Z    +0.000, E1   -23.548, E3 +492771.277}
SPL {X  -162.820, Y  +432.946, Z    +0.000, E1   -22.795, E3 +492785.681}
SPL {X  -162.820, Y  +434.888, Z    +0.000, E1   -22.823, E3 +492795.087}
SPL {X  -162.820, Y  +436.834, Z    +0.000, E1   -22.779, E3 +492805.048}
SPL {X  -162.820, Y  +438.868, Z    +0.000, E1   -22.837, E3 +492814.701}
SPL {X  -162.820, Y  +441.351, Z    +0.000, E1   -22.805, E3 +492827.276}
SPL {X  -162.820, Y  +443.809, Z    +0.000, E1   -22.804, E3 +492839.443}
SPL {X  -162.820, Y  +446.105, Z    +0.000, E1   -22.815, E3 +492850.685}
SPL {X  -162.820, Y  +447.974, Z    +0.000, E1   -22.856, E3 +492859.588}
SPL {X  -162.820, Y  +449.911, Z    +0.000, E1   -22.774, E3 +492869.863}
SPL {X  -162.820, Y  +451.861, Z    +0.000, E1   -22.750, E3 +492879.710}
SPL {X  -162.820, Y  +454.167, Z    +0.000, E1   -22.842, E3 +492890.440}
SPL {X  -162.820, Y  +456.529, Z    +0.000, E1   -22.855, E3 +492901.968}
SPL {X  -162.820, Y  +458.725, Z    +0.000, E1   -22.793, E3 +492913.372}
SPL {X  -162.820, Y  +461.700, Z    +0.000, E1   -22.822, E3 +492927.995}
SPL {X  -162.820, Y  +464.633, Z    +0.000, E1   -22.813, E3 +492942.492}
SPL {X  -162.820, Y  +466.699, Z    +0.000, E1   -22.824, E3 +492952.538}
SPL {X  -162.820, Y  +468.655, Z    +0.000, E1   -22.858, E3 +492961.981}
SPL {X  -162.820, Y  +470.892, Z    +0.000, E1   -22.837, E3 +492973.220}
SPL {X  -162.820, Y  +473.485, Z    +0.000, E1   -22.806, E3 +492986.419}
SPL {X  -162.820, Y  +475.738, Z    +0.000, E1   -22.728, E3 +492998.084}
SPL {X  -162.820, Y  +478.177, Z    +0.000, E1   -22.834, E3 +493009.423}
SPL {X  -162.820, Y  +481.034, Z    +0.000, E1   -22.831, E3 +493023.561}
SPL {X  -162.820, Y  +483.391, Z    +0.000, E1   -22.793, E3 +493035.497}
SPL {X  -162.820, Y  +486.307, Z    +0.000, E1   -22.833, E3 +493049.751}
SPL {X  -162.820, Y  +489.750, Z    +0.000, E1   -22.832, E3 +493066.821}
SPL {X  -162.820, Y  +493.233, Z    +0.000, E1   -22.844, E3 +493083.957}
SPL {X  -162.820, Y  +496.150, Z    +0.000, E1   -22.796, E3 +493098.677}
SPL {X  -162.820, Y  +498.661, Z    +0.000, E1   -22.828, E3 +493110.858}
SPL {X  -162.820, Y  +501.761, Z    +0.000, E1   -22.820, E3 +493126.426}
SPL {X  -162.820, Y  +505.323, Z    +0.000, E1   -22.838, E3 +493143.873}
SPL {X  -162.820, Y  +507.875, Z    +0.000, E1   -22.849, E3 +493156.241}
SPL {X  -162.820, Y  +510.068, Z    +0.000, E1   -22.761, E3 +493167.934}
SPL {X  -162.820, Y  +512.359, Z    +0.000, E1   -22.823, E3 +493178.665}
SPL {X  -162.820, Y  +514.562, Z    +0.000, E1   -22.806, E3 +493189.852}
SPL {X  -162.820, Y  +517.952, Z    +0.000, E1   -22.864, E3 +493206.250}
SPL {X  -162.820, Y  +520.641, Z    +0.000, E1   -22.790, E3 +493219.968}
SPL {X  -162.820, Y  +522.740, Z    +0.000, E1   -22.811, E3 +493230.210}
SPL {X  -162.820, Y  +524.628, Z    +0.000, E1   -22.846, E3 +493239.205}
SPL {X  -162.820, Y  +526.661, Z    +0.000, E1   -22.801, E3 +493249.761}
SPL {X  -162.820, Y  +529.662, Z    +0.000, E1   -22.810, E3 +493264.611}
SPL {X  -162.820, Y  +532.614, Z    +0.000, E1   -22.828, E3 +493279.018}
SPL {X  -162.820, Y  +534.838, Z    +0.000, E1   -22.864, E3 +493289.647}
SPL {X  -162.820, Y  +536.882, Z    +0.000, E1   -22.782, E3 +493300.502}
SPL {X  -162.820, Y  +539.194, Z    +0.000, E1   -22.826, E3 +493311.550}
SPL {X  -162.820, Y  +541.555, Z    +0.000, E1   -22.817, E3 +493323.364}
SPL {X  -162.820, Y  +543.728, Z    +0.000, E1   -22.799, E3 +493334.222}
SPL {X  -162.820, Y  +545.925, Z    +0.000, E1   -22.803, E3 +493345.092}
SPL {X  -162.820, Y  +548.328, Z    +0.000, E1   -22.796, E3 +493357.087}
SPL {X  -162.820, Y  +551.027, Z    +0.000, E1   -22.819, E3 +493370.280}
SPL {X  -162.820, Y  +553.721, Z    +0.000, E1   -22.807, E3 +493383.724}
SPL {X  -162.820, Y  +556.430, Z    +0.000, E1   -22.821, E3 +493397.020}
SPL {X  -162.820, Y  +558.974, Z    +0.000, E1   -22.806, E3 +493409.720}
SPL {X  -162.820, Y  +562.171, Z    +0.000, E1   -22.845, E3 +493425.418}
SPL {X  -162.820, Y  +565.170, Z    +0.000, E1   -22.801, E3 +493440.432}
SPL {X  -162.820, Y  +567.308, Z    +0.000, E1   -22.750, E3 +493451.448}
SPL {X  -162.820, Y  +570.378, Z    +0.000, E1   -22.843, E3 +493466.072}
SPL {X  -162.820, Y  +573.634, Z    +0.000, E1   -22.827, E3 +493482.215}
SPL {X  -162.820, Y  +576.228, Z    +0.000, E1   -22.814, E3 +493495.112}
SPL {X  -162.820, Y  +578.553, Z    +0.000, E1   -22.801, E3 +493506.728}
SPL {X  -162.820, Y  +581.064, Z    +0.000, E1   -22.823, E3 +493519.012}
SPL {X  -162.820, Y  +583.435, Z    +0.000, E1   -22.808, E3 +493530.834}
SPL {X  -162.820, Y  +585.410, Z    +0.000, E1   -22.764, E3 +493540.970}
SPL {X  -162.820, Y  +587.676, Z    +0.000, E1   -22.853, E3 +493551.484}
SPL {X  -162.820, Y  +590.707, Z    +0.000, E1   -22.855, E3 +493566.634}
SPL {X  -162.820, Y  +593.650, Z    +0.000, E1   -22.810, E3 +493581.395}
SPL {X  -162.820, Y  +595.830, Z    +0.000, E1   -22.828, E3 +493592.010}
SPL {X  -162.820, Y  +598.094, Z    +0.000, E1   -22.843, E3 +493603.124}
SPL {X  -162.820, Y  +600.420, Z    +0.000, E1   -22.826, E3 +493614.755}
SPL {X  -162.820, Y  +602.573, Z    +0.000, E1   -22.830, E3 +493625.340}
SPL {X  -162.820, Y  +604.828, Z    +0.000, E1   -22.784, E3 +493636.978}
SPL {X  -162.820, Y  +608.133, Z    +0.000, E1   -22.831, E3 +493653.096}
SPL {X  -162.820, Y  +611.103, Z    +0.000, E1   -22.785, E3 +493668.022}
SPL {X  -162.820, Y  +613.294, Z    +0.000, E1   -22.780, E3 +493678.895}
SPL {X  -162.820, Y  +615.356, Z    +0.000, E1   -22.799, E3 +493688.952}
SPL {X  -162.820, Y  +617.439, Z    +0.000, E1   -22.808, E3 +493699.210}
SPL {X  -162.820, Y  +619.665, Z    +0.000, E1   -22.817, E3 +493710.178}
SPL {X  -162.820, Y  +621.733, Z    +0.000, E1   -22.759, E3 +493720.903}
SPL {X  -162.820, Y  +624.076, Z    +0.000, E1   -22.774, E3 +493732.408}
SPL {X  -162.820, Y  +626.527, Z    +0.000, E1   -22.768, E3 +493744.650}
SPL {X  -162.820, Y  +629.758, Z    +0.000, E1   -22.800, E3 +493760.579}
SPL {X  -162.820, Y  +632.572, Z    +0.000, E1   -22.785, E3 +493774.428}
SPL {X  -162.820, Y  +634.507, Z    +0.000, E1   -22.784, E3 +493784.067}
SPL {X  -162.820, Y  +636.863, Z    +0.000, E1   -22.760, E3 +493795.989}
SPL {X  -162.820, Y  +639.254, Z    +0.000, E1   -22.767, E3 +493807.773}
SPL {X  -162.820, Y  +641.888, Z    +0.000, E1   -22.790, E3 +493820.720}
SPL {X  -162.820, Y  +644.915, Z    +0.000, E1   -22.818, E3 +493835.495}
SPL {X  -162.820, Y  +647.561, Z    +0.000, E1   -22.705, E3 +493849.537}
SPL {X  -162.820, Y  +649.758, Z    +0.000, E1   -22.780, E3 +493859.727}
SPL {X  -162.820, Y  +651.708, Z    +0.000, E1   -22.810, E3 +493869.221}
SPL {X  -162.820, Y  +653.898, Z    +0.000, E1   -22.796, E3 +493880.142}
SPL {X  -162.820, Y  +656.161, Z    +0.000, E1   -22.812, E3 +493891.264}
SPL {X  -162.820, Y  +658.384, Z    +0.000, E1   -22.822, E3 +493902.130}
SPL {X  -162.820, Y  +660.215, Z    +0.000, E1   -22.649, E3 +493912.720}
SPL {X  -162.820, Y  +662.823, Z    +0.000, E1   -22.799, E3 +493924.428}
SPL {X  -162.820, Y  +665.862, Z    +0.000, E1   -22.864, E3 +493939.128}
SPL {X  -162.820, Y  +668.960, Z    +0.000, E1   -22.773, E3 +493955.079}
SPL {X  -162.820, Y  +671.605, Z    +0.000, E1   -22.777, E3 +493968.152}
SPL {X  -162.817, Y  +674.515, Z    +0.000, E1   -22.816, E3 +493982.349}
SPL {X  -162.773, Y  +677.428, Z    +0.000, E1   -22.762, E3 +493997.157}
SPL {X  -162.691, Y  +679.987, Z    +0.000, E1   -22.794, E3 +494009.571}
SPL {X  -162.559, Y  +682.717, Z    +0.000, E1   -22.726, E3 +494023.754}
SPL {X  -162.404, Y  +685.137, Z    +0.000, E1   -22.766, E3 +494035.276}
SPL {X  -162.229, Y  +687.364, Z    +0.000, E1   -22.685, E3 +494047.145}
SPL {X  -161.938, Y  +690.422, Z    +0.000, E1   -22.769, E3 +494061.551}
SPL {X  -161.065, Y  +697.344, Z    +0.000, E1   -25.698, E3 +494070.670}
SPL {X  -158.553, Y  +710.529, Z    +0.000, E1   -30.890, E3 +494084.567}
ENDSPLINE

SPLINE
SPL {X  -161.215, Y  +696.305, Z    +0.000, E1   -20.575, E3 +494111.148}
SPL {X  -161.691, Y  +692.643, Z    +0.000, E1   -17.369, E3 +494127.336}
SPL {X  -162.534, Y  +683.153, Z    +0.000, E1   -10.475, E3 +494152.803}
SPL {X  -162.820, Y  +667.630, Z    +0.000, E1    -0.882, E3 +494146.779}
SPL {X  -162.820, Y  +661.883, Z    +0.000, E1    +3.373, E3 +494152.223}
SPL {X  -162.820, Y  +655.163, Z    +0.000, E1    +8.702, E3 +494151.821}
SPL {X  -162.820, Y  +634.515, Z    +0.000, E1   +26.439, E3 +494144.235}
ENDSPLINE

SPLINE
SPL {X  -162.820, Y  +638.080, Z    +0.000, E1   +18.858, E3 +494174.199}
ENDSPLINE

SPLINE
SPL {X  -162.820, Y  +623.278, Z    +0.000, E1   +28.723, E3 +494175.770}
SPL {X  -162.820, Y  +618.658, Z    +0.000, E1   +26.841, E3 +494204.378}
ENDSPLINE

SPLINE
SPL {X  -162.820, Y  +623.685, Z    +0.000, E1   +22.346, E3 +494216.685}
ENDSPLINE

SPLINE
SPL {X  -162.820, Y  +621.304, Z    +0.000, E1   +22.259, E3 +494229.500}
SPL {X  -162.820, Y  +618.758, Z    +0.000, E1   +22.239, E3 +494242.651}
SPL {X  -162.820, Y  +616.062, Z    +0.000, E1   +22.275, E3 +494256.072}
SPL {X  -162.820, Y  +613.536, Z    +0.000, E1   +22.242, E3 +494269.193}
SPL {X  -162.820, Y  +611.128, Z    +0.000, E1   +22.252, E3 +494281.364}
SPL {X  -162.820, Y  +608.428, Z    +0.000, E1   +22.255, E3 +494295.147}
SPL {X  -162.820, Y  +605.984, Z    +0.000, E1   +22.221, E3 +494307.784}
SPL {X  -162.820, Y  +603.020, Z    +0.000, E1   +22.272, E3 +494322.683}
SPL {X  -162.820, Y  +599.842, Z    +0.000, E1   +22.298, E3 +494338.448}
SPL {X  -162.820, Y  +597.194, Z    +0.000, E1   +22.253, E3 +494352.369}
SPL {X  -162.820, Y  +594.779, Z    +0.000, E1   +22.284, E3 +494364.273}
SPL {X  -162.820, Y  +592.389, Z    +0.000, E1   +22.245, E3 +494376.890}
SPL {X  -162.820, Y  +589.492, Z    +0.000, E1   +22.304, E3 +494391.074}
SPL {X  -162.820, Y  +587.447, Z    +0.000, E1   +22.279, E3 +494401.603}
SPL {X  -162.820, Y  +585.192, Z    +0.000, E1   +22.298, E3 +494413.013}
SPL {X  -162.820, Y  +582.610, Z    +0.000, E1   +22.234, E3 +494426.637}
SPL {X  -162.820, Y  +580.317, Z    +0.000, E1   +22.300, E3 +494437.690}
SPL {X  -162.820, Y  +578.878, Z    +0.000, E1   +22.272, E3 +494445.200}
SPL {X  -162.820, Y  +576.856, Z    +0.000, E1   +22.233, E3 +494455.958}
SPL {X  -162.820, Y  +574.811, Z    +0.000, E1   +22.236, E3 +494466.222}
SPL {X  -162.820, Y  +572.645, Z    +0.000, E1   +22.246, E3 +494477.317}
SPL {X  -162.820, Y  +569.475, Z    +0.000, E1   +22.269, E3 +494493.324}
SPL {X  -162.820, Y  +565.838, Z    +0.000, E1   +22.271, E3 +494511.918}
SPL {X  -162.820, Y  +562.162, Z    +0.000, E1   +22.252, E3 +494530.735}
SPL {X  -162.820, Y  +558.919, Z    +0.000, E1   +22.286, E3 +494546.899}
SPL {X  -162.820, Y  +556.169, Z    +0.000, E1   +22.295, E3 +494560.728}
SPL {X  -162.820, Y  +553.294, Z    +0.000, E1   +22.266, E3 +494575.726}
SPL {X  -162.820, Y  +550.136, Z    +0.000, E1   +22.258, E3 +494591.839}
SPL {X  -162.820, Y  +546.694, Z    +0.000, E1   +22.290, E3 +494609.161}
SPL {X  -162.820, Y  +543.558, Z    +0.000, E1   +22.285, E3 +494625.024}
SPL {X  -162.820, Y  +541.633, Z    +0.000, E1   +22.257, E3 +494634.952}
SPL {X  -162.820, Y  +539.116, Z    +0.000, E1   +22.302, E3 +494647.563}
SPL {X  -162.820, Y  +536.913, Z    +0.000, E1   +22.192, E3 +494659.487}
SPL {X  -162.820, Y  +534.880, Z    +0.000, E1   +22.252, E3 +494669.441}
SPL {X  -162.820, Y  +532.896, Z    +0.000, E1   +22.234, E3 +494679.601}
SPL {X  -162.820, Y  +531.056, Z    +0.000, E1   +22.251, E3 +494688.883}
SPL {X  -162.820, Y  +528.708, Z    +0.000, E1   +22.319, E3 +494700.265}
SPL {X  -162.820, Y  +525.932, Z    +0.000, E1   +22.258, E3 +494715.021}
SPL {X  -162.820, Y  +522.524, Z    +0.000, E1   +22.326, E3 +494731.745}
SPL {X  -162.820, Y  +519.457, Z    +0.000, E1   +22.481, E3 +494745.874}
SPL {X  -162.820, Y  +506.285, Z    +0.000, E1   +28.538, E3 +494757.332}
SPL {X  -162.820, Y  +504.441, Z    +0.000, E1   +27.574, E3 +494771.674}
SPL {X  -162.820, Y  +502.813, Z    +0.000, E1   +26.013, E3 +494789.871}
SPL {X  -162.820, Y  +502.016, Z    +0.000, E1   +24.802, E3 +494802.214}
SPL {X  -162.820, Y  +501.060, Z    +0.000, E1   +24.081, E3 +494812.404}
SPL {X  -162.820, Y  +499.934, Z    +0.000, E1   +22.814, E3 +494828.272}
SPL {X  -162.820, Y  +498.303, Z    +0.000, E1   +21.749, E3 +494845.528}
SPL {X  -162.820, Y  +495.897, Z    +0.000, E1   +21.662, E3 +494858.682}
SPL {X  -162.820, Y  +493.717, Z    +0.000, E1   +21.704, E3 +494869.788}
SPL {X  -162.820, Y  +491.396, Z    +0.000, E1   +21.707, E3 +494881.912}
SPL {X  -162.820, Y  +489.485, Z    +0.000, E1   +21.661, E3 +494892.260}
SPL {X  -162.820, Y  +487.723, Z    +0.000, E1   +21.665, E3 +494901.463}
SPL {X  -162.820, Y  +485.661, Z    +0.000, E1   +21.712, E3 +494911.907}
SPL {X  -162.820, Y  +482.775, Z    +0.000, E1   +21.716, E3 +494927.159}
SPL {X  -162.820, Y  +479.894, Z    +0.000, E1   +21.695, E3 +494942.236}
SPL {X  -162.820, Y  +477.685, Z    +0.000, E1   +21.656, E3 +494954.173}
SPL {X  -162.820, Y  +475.419, Z    +0.000, E1   +21.711, E3 +494965.526}
SPL {X  -162.820, Y  +473.301, Z    +0.000, E1   +21.712, E3 +494976.623}
SPL {X  -162.820, Y  +470.965, Z    +0.000, E1   +21.700, E3 +494988.968}
SPL {X  -162.820, Y  +469.036, Z    +0.000, E1   +21.695, E3 +494999.012}
SPL {X  -162.820, Y  +467.138, Z    +0.000, E1   +21.678, E3 +495009.183}
SPL {X  -162.820, Y  +465.011, Z    +0.000, E1   +21.692, E3 +495020.166}
SPL {X  -162.820, Y  +462.669, Z    +0.000, E1   +21.752, E3 +495031.946}
SPL {X  -162.820, Y  +460.725, Z    +0.000, E1   +21.689, E3 +495042.559}
SPL {X  -162.820, Y  +458.666, Z    +0.000, E1   +21.695, E3 +495053.371}
SPL {X  -162.820, Y  +456.431, Z    +0.000, E1   +21.708, E3 +495064.900}
SPL {X  -162.820, Y  +454.628, Z    +0.000, E1   +21.674, E3 +495074.618}
SPL {X  -162.820, Y  +452.690, Z    +0.000, E1   +21.773, E3 +495083.892}
SPL {X  -162.820, Y  +450.610, Z    +0.000, E1   +21.698, E3 +495095.491}
SPL {X  -162.820, Y  +448.170, Z    +0.000, E1   +21.667, E3 +495108.512}
SPL {X  -162.820, Y  +446.246, Z    +0.000, E1   +21.696, E3 +495118.330}
SPL {X  -162.820, Y  +443.784, Z    +0.000, E1   +21.713, E3 +495131.116}
SPL {X  -162.820, Y  +441.754, Z    +0.000, E1   +21.708, E3 +495141.668}
SPL {X  -162.820, Y  +439.933, Z    +0.000, E1   +21.690, E3 +495151.432}
SPL {X  -162.820, Y  +437.628, Z    +0.000, E1   +21.678, E3 +495163.620}
SPL {X  -162.820, Y  +435.262, Z    +0.000, E1   +21.727, E3 +495175.555}
SPL {X  -162.820, Y  +433.510, Z    +0.000, E1   +21.692, E3 +495184.969}
SPL {X  -162.820, Y  +431.492, Z    +0.000, E1   +21.686, E3 +495195.665}
SPL {X  -162.820, Y  +429.074, Z    +0.000, E1   +21.710, E3 +495208.116}
SPL {X  -162.820, Y  +427.020, Z    +0.000, E1   +21.674, E3 +495219.118}
SPL {X  -162.820, Y  +424.525, Z    +0.000, E1   +21.712, E3 +495232.031}
SPL {X  -162.820, Y  +421.144, Z    +0.000, E1   +21.719, E3 +495249.698}
SPL {X  -162.820, Y  +418.116, Z    +0.000, E1   +21.761, E3 +495265.029}
SPL {X  -162.820, Y  +416.127, Z    +0.000, E1   +21.715, E3 +495275.734}
SPL {X  -162.820, Y  +414.361, Z    +0.000, E1   +21.613, E3 +495285.921}
SPL {X  -162.820, Y  +412.134, Z    +0.000, E1   +21.697, E3 +495296.866}
SPL {X  -162.820, Y  +409.248, Z    +0.000, E1   +21.741, E3 +495311.801}
SPL {X  -162.820, Y  +406.238, Z    +0.000, E1   +21.697, E3 +495327.769}
SPL {X  -162.820, Y  +404.001, Z    +0.000, E1   +21.723, E3 +495339.199}
SPL {X  -162.820, Y  +402.223, Z    +0.000, E1   +21.697, E3 +495348.684}
SPL {X  -162.820, Y  +400.348, Z    +0.000, E1   +21.713, E3 +495358.410}
SPL {X  -162.820, Y  +398.298, Z    +0.000, E1   +21.721, E3 +495369.026}
SPL {X  -162.820, Y  +396.371, Z    +0.000, E1   +21.713, E3 +495379.208}
SPL {X  -162.820, Y  +394.508, Z    +0.000, E1   +21.616, E3 +495389.763}
SPL {X  -162.820, Y  +392.435, Z    +0.000, E1   +21.681, E3 +495400.116}
SPL {X  -162.820, Y  +389.390, Z    +0.000, E1   +21.742, E3 +495415.723}
SPL {X  -162.820, Y  +386.818, Z    +0.000, E1   +21.679, E3 +495429.482}
SPL {X  -162.820, Y  +384.697, Z    +0.000, E1   +21.693, E3 +495440.552}
SPL {X  -162.820, Y  +382.288, Z    +0.000, E1   +21.742, E3 +495452.676}
SPL {X  -162.820, Y  +380.381, Z    +0.000, E1   +21.655, E3 +495463.401}
SPL {X  -162.808, Y  +378.512, Z    +0.000, E1   +21.736, E3 +495472.453}
SPL {X  -162.776, Y  +376.710, Z    +0.000, E1   +21.698, E3 +495482.252}
SPL {X  -162.707, Y  +374.438, Z    +0.000, E1   +21.688, E3 +495494.256}
SPL {X  -162.607, Y  +372.171, Z    +0.000, E1   +21.692, E3 +495506.056}
SPL {X  -162.494, Y  +370.197, Z    +0.000, E1   +21.655, E3 +495516.682}
SPL {X  -162.349, Y  +368.131, Z    +0.000, E1   +21.624, E3 +495527.800}
SPL {X  -162.161, Y  +365.866, Z    +0.000, E1   +21.642, E3 +495539.485}
SPL {X  -161.927, Y  +363.466, Z    +0.000, E1   +21.730, E3 +495551.257}
SPL {X  -160.290, Y  +351.907, Z    +0.000, E1   +27.562, E3 +495558.835}
SPL {X  -159.725, Y  +348.905, Z    +0.000, E1   +26.136, E3 +495584.070}
ENDSPLINE

SPLINE
SPL {X  -160.871, Y  +355.385, Z    +0.000, E1   +21.841, E3 +495592.913}
SPL {X  -161.833, Y  +362.603, Z    +0.000, E1   +17.021, E3 +495602.944}
ENDSPLINE

SPLINE
SPL {X  -160.786, Y  +354.842, Z    +0.000, E1   +19.274, E3 +495635.099}
ENDSPLINE

SPLINE
SPL {X  -162.485, Y  +370.062, Z    +0.000, E1   +10.606, E3 +495641.477}
SPL {X  -162.820, Y  +381.311, Z    +0.000, E1    +4.054, E3 +495631.833}
SPL {X  -162.820, Y  +389.994, Z    +0.000, E1    -2.149, E3 +495626.245}
SPL {X  -162.820, Y  +391.982, Z    +0.000, E1    -3.443, E3 +495636.690}
SPL {X  -162.820, Y  +399.630, Z    +0.000, E1    -9.426, E3 +495639.198}
SPL {X  -162.820, Y  +408.127, Z    +0.000, E1   -18.417, E3 +495625.486}
SPL {X  -162.820, Y  +420.083, Z    +0.000, E1   -24.325, E3 +495645.961}
SPL {X  -162.820, Y  +428.527, Z    +0.000, E1   -26.988, E3 +495663.254}
SPL {X  -162.820, Y  +431.191, Z    +0.000, E1   -23.548, E3 +495698.107}
SPL {X  -162.820, Y  +432.946, Z    +0.000, E1   -22.795, E3 +495712.510}
SPL {X  -162.820, Y  +434.888, Z    +0.000, E1   -22.823, E3 +495721.917}
SPL {X  -162.820, Y  +436.834, Z    +0.000, E1   -22.779, E3 +495731.877}
SPL {X  -162.820, Y  +438.868, Z    +0.000, E1   -22.837, E3 +495741.530}
SPL {X  -162.820, Y  +441.351, Z    +0.000, E1   -22.805, E3 +495754.106}
SPL {X  -162.820, Y  +443.809, Z    +0.000, E1   -22.804, E3 +495766.272}
SPL {X  -162.820, Y  +446.105, Z    +0.000, E1   -22.815, E3 +495777.514}
SPL {X  -162.820, Y  +447.974, Z    +0.000, E1   -22.856, E3 +495786.417}
SPL {X  -162.820, Y  +449.911, Z    +0.000, E1   -22.774, E3 +495796.692}
SPL {X  -162.820, Y  +451.861, Z    +0.000, E1   -22.750, E3 +495806.539}
SPL {X  -162.820, Y  +454.167, Z    +0.000, E1   -22.842, E3 +495817.269}
SPL {X  -162.820, Y  +456.529, Z    +0.000, E1   -22.855, E3 +495828.797}
SPL {X  -162.820, Y  +458.725, Z    +0.000, E1   -22.793, E3 +495840.202}
SPL {X  -162.820, Y  +461.700, Z    +0.000, E1   -22.822, E3 +495854.824}
SPL {X  -162.820, Y  +464.633, Z    +0.000, E1   -22.813, E3 +495869.321}
SPL {X  -162.820, Y  +466.699, Z    +0.000, E1   -22.824, E3 +495879.367}
SPL {X  -162.820, Y  +468.655, Z    +0.000, E1   -22.858, E3 +495888.811}
SPL {X  -162.820, Y  +470.892, Z    +0.000, E1   -22.837, E3 +495900.049}
SPL {X  -162.820, Y  +473.485, Z    +0.000, E1   -22.806, E3 +495913.248}
SPL {X  -162.820, Y  +475.738, Z    +0.000, E1   -22.728, E3 +495924.913}
SPL {X  -162.820, Y  +478.177, Z    +0.000, E1   -22.834, E3 +495936.252}
SPL {X  -162.820, Y  +481.034, Z    +0.000, E1   -22.831, E3 +495950.390}
SPL {X  -162.820, Y  +483.391, Z    +0.000, E1   -22.793, E3 +495962.326}
SPL {X  -162.820, Y  +486.307, Z    +0.000, E1   -22.833, E3 +495976.580}
SPL {X  -162.820, Y  +489.750, Z    +0.000, E1   -22.832, E3 +495993.650}
SPL {X  -162.820, Y  +493.233, Z    +0.000, E1   -22.844, E3 +496010.787}
SPL {X  -162.820, Y  +496.150, Z    +0.000, E1   -22.796, E3 +496025.506}
SPL {X  -162.820, Y  +498.661, Z    +0.000, E1   -22.828, E3 +496037.687}
SPL {X  -162.820, Y  +501.761, Z    +0.000, E1   -22.820, E3 +496053.256}
SPL {X  -162.820, Y  +505.323, Z    +0.000, E1   -22.838, E3 +496070.702}
SPL {X  -162.820, Y  +507.875, Z    +0.000, E1   -22.849, E3 +496083.070}
SPL {X  -162.820, Y  +510.068, Z    +0.000, E1   -22.761, E3 +496094.763}
SPL {X  -162.820, Y  +512.359, Z    +0.000, E1   -22.823, E3 +496105.494}
SPL {X  -162.820, Y  +514.562, Z    +0.000, E1   -22.806, E3 +496116.681}
SPL {X  -162.820, Y  +517.952, Z    +0.000, E1   -22.864, E3 +496133.079}
SPL {X  -162.820, Y  +520.641, Z    +0.000, E1   -22.790, E3 +496146.797}
SPL {X  -162.820, Y  +522.740, Z    +0.000, E1   -22.811, E3 +496157.040}
SPL {X  -162.820, Y  +524.628, Z    +0.000, E1   -22.846, E3 +496166.035}
SPL {X  -162.820, Y  +526.661, Z    +0.000, E1   -22.801, E3 +496176.590}
SPL {X  -162.820, Y  +529.662, Z    +0.000, E1   -22.810, E3 +496191.441}
SPL {X  -162.820, Y  +532.614, Z    +0.000, E1   -22.828, E3 +496205.847}
SPL {X  -162.820, Y  +534.838, Z    +0.000, E1   -22.864, E3 +496216.476}
SPL {X  -162.820, Y  +536.882, Z    +0.000, E1   -22.782, E3 +496227.331}
SPL {X  -162.820, Y  +539.194, Z    +0.000, E1   -22.826, E3 +496238.379}
SPL {X  -162.820, Y  +541.555, Z    +0.000, E1   -22.817, E3 +496250.194}
SPL {X  -162.820, Y  +543.728, Z    +0.000, E1   -22.799, E3 +496261.051}
SPL {X  -162.820, Y  +545.925, Z    +0.000, E1   -22.803, E3 +496271.921}
SPL {X  -162.820, Y  +548.328, Z    +0.000, E1   -22.796, E3 +496283.917}
SPL {X  -162.820, Y  +551.027, Z    +0.000, E1   -22.819, E3 +496297.109}
SPL {X  -162.820, Y  +553.721, Z    +0.000, E1   -22.807, E3 +496310.554}
SPL {X  -162.820, Y  +556.430, Z    +0.000, E1   -22.821, E3 +496323.850}
SPL {X  -162.820, Y  +559.675, Z    +0.000, E1   -22.837, E3 +496339.930}
SPL {X  -162.820, Y  +562.799, Z    +0.000, E1   -22.814, E3 +496355.436}
SPL {X  -162.820, Y  +565.170, Z    +0.000, E1   -22.801, E3 +496367.261}
SPL {X  -162.820, Y  +568.020, Z    +0.000, E1   -22.787, E3 +496381.648}
SPL {X  -162.820, Y  +570.992, Z    +0.000, E1   -22.834, E3 +496395.867}
SPL {X  -162.820, Y  +572.901, Z    +0.000, E1   -22.775, E3 +496405.735}
SPL {X  -162.820, Y  +575.638, Z    +0.000, E1   -22.855, E3 +496418.845}
SPL {X  -162.820, Y  +578.553, Z    +0.000, E1   -22.801, E3 +496433.557}
SPL {X  -162.820, Y  +581.064, Z    +0.000, E1   -22.823, E3 +496445.841}
SPL {X  -162.820, Y  +583.435, Z    +0.000, E1   -22.808, E3 +496457.663}
SPL {X  -162.820, Y  +585.410, Z    +0.000, E1   -22.764, E3 +496467.799}
SPL {X  -162.820, Y  +587.676, Z    +0.000, E1   -22.853, E3 +496478.313}
SPL {X  -162.820, Y  +589.682, Z    +0.000, E1   -22.776, E3 +496488.843}
SPL {X  -162.820, Y  +591.720, Z    +0.000, E1   -22.868, E3 +496498.154}
SPL {X  -162.820, Y  +593.650, Z    +0.000, E1   -22.810, E3 +496508.224}
SPL {X  -162.820, Y  +595.830, Z    +0.000, E1   -22.828, E3 +496518.840}
SPL {X  -162.820, Y  +598.094, Z    +0.000, E1   -22.843, E3 +496529.953}
SPL {X  -162.820, Y  +600.420, Z    +0.000, E1   -22.826, E3 +496541.584}
SPL {X  -162.820, Y  +602.573, Z    +0.000, E1   -22.830, E3 +496552.169}
SPL {X  -162.820, Y  +604.828, Z    +0.000, E1   -22.784, E3 +496563.808}
SPL {X  -162.820, Y  +608.133, Z    +0.000, E1   -22.831, E3 +496579.925}
SPL {X  -162.820, Y  +611.103, Z    +0.000, E1   -22.785, E3 +496594.851}
SPL {X  -162.820, Y  +613.294, Z    +0.000, E1   -22.780, E3 +496605.724}
SPL {X  -162.820, Y  +615.356, Z    +0.000, E1   -22.799, E3 +496615.782}
SPL {X  -162.820, Y  +617.439, Z    +0.000, E1   -22.808, E3 +496626.040}
SPL {X  -162.820, Y  +619.665, Z    +0.000, E1   -22.817, E3 +496637.008}
SPL {X  -162.820, Y  +621.733, Z    +0.000, E1   -22.759, E3 +496647.732}
SPL {X  -162.820, Y  +624.076, Z    +0.000, E1   -22.774, E3 +496659.237}
SPL {X  -162.820, Y  +627.244, Z    +0.000, E1   -22.803, E3 +496674.919}
SPL {X  -162.820, Y  +630.349, Z    +0.000, E1   -22.766, E3 +496690.451}
SPL {X  -162.820, Y  +632.572, Z    +0.000, E1   -22.785, E3 +496701.258}
SPL {X  -162.820, Y  +634.507, Z    +0.000, E1   -22.784, E3 +496710.897}
SPL {X  -162.820, Y  +636.863, Z    +0.000, E1   -22.760, E3 +496722.819}
SPL {X  -162.820, Y  +640.111, Z    +0.000, E1   -22.809, E3 +496738.702}
SPL {X  -162.820, Y  +643.449, Z    +0.000, E1   -22.796, E3 +496755.219}
SPL {X  -162.820, Y  +645.630, Z    +0.000, E1   -22.795, E3 +496765.915}
SPL {X  -162.820, Y  +647.561, Z    +0.000, E1   -22.705, E3 +496776.366}
SPL {X  -162.820, Y  +651.051, Z    +0.000, E1   -22.833, E3 +496792.785}
SPL {X  -162.820, Y  +653.898, Z    +0.000, E1   -22.796, E3 +496806.971}
SPL {X  -162.820, Y  +656.161, Z    +0.000, E1   -22.812, E3 +496818.093}
SPL {X  -162.820, Y  +658.384, Z    +0.000, E1   -22.822, E3 +496828.959}
SPL {X  -162.820, Y  +660.215, Z    +0.000, E1   -22.649, E3 +496839.550}
SPL {X  -162.820, Y  +662.823, Z    +0.000, E1   -22.799, E3 +496851.258}
SPL {X  -162.820, Y  +665.112, Z    +0.000, E1   -22.835, E3 +496862.312}
SPL {X  -162.820, Y  +667.016, Z    +0.000, E1   -22.823, E3 +496871.740}
SPL {X  -162.820, Y  +668.960, Z    +0.000, E1   -22.773, E3 +496881.908}
SPL {X  -162.820, Y  +672.333, Z    +0.000, E1   -22.837, E3 +496898.244}
SPL {X  -162.812, Y  +675.071, Z    +0.000, E1   -22.742, E3 +496912.389}
SPL {X  -162.773, Y  +677.428, Z    +0.000, E1   -22.762, E3 +496923.987}
SPL {X  -162.691, Y  +679.987, Z    +0.000, E1   -22.794, E3 +496936.400}
SPL {X  -162.559, Y  +682.717, Z    +0.000, E1   -22.726, E3 +496950.583}
SPL {X  -162.404, Y  +685.137, Z    +0.000, E1   -22.766, E3 +496962.106}
SPL {X  -162.229, Y  +687.364, Z    +0.000, E1   -22.685, E3 +496973.974}
SPL {X  -161.938, Y  +690.422, Z    +0.000, E1   -22.769, E3 +496988.380}
SPL {X  -161.065, Y  +697.344, Z    +0.000, E1   -25.698, E3 +496997.500}
SPL {X  -158.730, Y  +709.763, Z    +0.000, E1   -31.225, E3 +497006.173}
ENDSPLINE

SPLINE
SPL {X  -160.932, Y  +698.225, Z    +0.000, E1   -21.712, E3 +497037.282}
SPL {X  -161.917, Y  +690.622, Z    +0.000, E1   -16.445, E3 +497050.883}
ENDSPLINE

SPLINE
SPL {X  -161.349, Y  +695.340, Z    +0.000, E1   -18.625, E3 +497058.502}
ENDSPLINE

SPLINE
SPL {X  -162.534, Y  +683.153, Z    +0.000, E1   -10.475, E3 +497079.632}
SPL {X  -162.820, Y  +667.630, Z    +0.000, E1    -0.882, E3 +497073.609}
SPL {X  -162.820, Y  +661.883, Z    +0.000, E1    +3.373, E3 +497079.052}
SPL {X  -162.820, Y  +655.163, Z    +0.000, E1    +8.702, E3 +497078.650}
SPL {X  -162.820, Y  +634.515, Z    +0.000, E1   +26.439, E3 +497071.064}
ENDSPLINE

SPLINE
SPL {X  -162.820, Y  +638.080, Z    +0.000, E1   +18.858, E3 +497101.028}
ENDSPLINE

SPLINE
SPL {X  -162.820, Y  +623.278, Z    +0.000, E1   +28.723, E3 +497102.599}
SPL {X  -162.820, Y  +618.658, Z    +0.000, E1   +26.841, E3 +497131.208}
ENDSPLINE

SPLINE
SPL {X  -162.820, Y  +623.685, Z    +0.000, E1   +22.346, E3 +497143.515}
ENDSPLINE

SPLINE
SPL {X  -162.820, Y  +621.304, Z    +0.000, E1   +22.259, E3 +497156.330}
SPL {X  -162.820, Y  +618.758, Z    +0.000, E1   +22.239, E3 +497169.480}
SPL {X  -162.820, Y  +616.062, Z    +0.000, E1   +22.275, E3 +497182.901}
SPL {X  -162.820, Y  +613.536, Z    +0.000, E1   +22.242, E3 +497196.023}
SPL {X  -162.820, Y  +611.128, Z    +0.000, E1   +22.252, E3 +497208.193}
SPL {X  -162.820, Y  +608.428, Z    +0.000, E1   +22.255, E3 +497221.977}
SPL {X  -162.820, Y  +605.178, Z    +0.000, E1   +22.267, E3 +497238.509}
SPL {X  -162.820, Y  +602.350, Z    +0.000, E1   +22.224, E3 +497253.126}
SPL {X  -162.820, Y  +599.168, Z    +0.000, E1   +22.310, E3 +497268.780}
SPL {X  -162.820, Y  +595.597, Z    +0.000, E1   +22.284, E3 +497287.116}
SPL {X  -162.820, Y  +593.320, Z    +0.000, E1   +22.199, E3 +497299.206}
SPL {X  -162.820, Y  +591.031, Z    +0.000, E1   +22.283, E3 +497310.297}
SPL {X  -162.820, Y  +588.026, Z    +0.000, E1   +22.301, E3 +497325.424}
SPL {X  -162.820, Y  +585.899, Z    +0.000, E1   +22.286, E3 +497336.226}
SPL {X  -162.820, Y  +583.204, Z    +0.000, E1   +22.278, E3 +497350.249}
SPL {X  -162.820, Y  +579.691, Z    +0.000, E1   +22.312, E3 +497367.737}
SPL {X  -162.820, Y  +577.460, Z    +0.000, E1   +22.218, E3 +497379.724}
SPL {X  -162.820, Y  +575.394, Z    +0.000, E1   +22.240, E3 +497390.149}
SPL {X  -162.820, Y  +572.645, Z    +0.000, E1   +22.246, E3 +497404.147}
SPL {X  -162.820, Y  +570.282, Z    +0.000, E1   +22.231, E3 +497416.197}
SPL {X  -162.820, Y  +567.961, Z    +0.000, E1   +22.247, E3 +497427.987}
SPL {X  -162.820, Y  +564.506, Z    +0.000, E1   +22.298, E3 +497445.301}
SPL {X  -162.820, Y  +561.620, Z    +0.000, E1   +22.191, E3 +497460.682}
SPL {X  -162.820, Y  +559.515, Z    +0.000, E1   +22.273, E3 +497470.684}
SPL {X  -162.820, Y  +556.723, Z    +0.000, E1   +22.309, E3 +497484.767}
SPL {X  -162.820, Y  +553.294, Z    +0.000, E1   +22.266, E3 +497502.555}
SPL {X  -162.820, Y  +550.136, Z    +0.000, E1   +22.258, E3 +497518.668}
SPL {X  -162.820, Y  +546.694, Z    +0.000, E1   +22.290, E3 +497535.990}
SPL {X  -162.820, Y  +543.558, Z    +0.000, E1   +22.285, E3 +497551.853}
SPL {X  -162.820, Y  +541.633, Z    +0.000, E1   +22.257, E3 +497561.781}
SPL {X  -162.820, Y  +539.116, Z    +0.000, E1   +22.302, E3 +497574.392}
SPL {X  -162.820, Y  +536.913, Z    +0.000, E1   +22.192, E3 +497586.316}
SPL {X  -162.820, Y  +534.880, Z    +0.000, E1   +22.252, E3 +497596.270}
SPL {X  -162.820, Y  +532.896, Z    +0.000, E1   +22.234, E3 +497606.430}
SPL {X  -162.820, Y  +531.056, Z    +0.000, E1   +22.251, E3 +497615.712}
SPL {X  -162.820, Y  +528.708, Z    +0.000, E1   +22.319, E3 +497627.094}
SPL {X  -162.820, Y  +525.932, Z    +0.000, E1   +22.258, E3 +497641.850}
SPL {X  -162.820, Y  +522.524, Z    +0.000, E1   +22.326, E3 +497658.574}
SPL {X  -162.820, Y  +519.457, Z    +0.000, E1   +22.481, E3 +497672.703}
SPL {X  -162.820, Y  +506.285, Z    +0.000, E1   +28.538, E3 +497684.161}
SPL {X  -162.820, Y  +504.441, Z    +0.000, E1   +27.574, E3 +497698.503}
SPL {X  -162.820, Y  +502.813, Z    +0.000, E1   +26.013, E3 +497716.701}
SPL {X  -162.820, Y  +502.016, Z    +0.000, E1   +24.802, E3 +497729.043}
SPL {X  -162.820, Y  +501.060, Z    +0.000, E1   +24.081, E3 +497739.233}
SPL {X  -162.820, Y  +499.934, Z    +0.000, E1   +22.814, E3 +497755.101}
SPL {X  -162.820, Y  +498.303, Z    +0.000, E1   +21.749, E3 +497772.358}
SPL {X  -162.820, Y  +495.897, Z    +0.000, E1   +21.662, E3 +497785.511}
SPL {X  -162.820, Y  +493.717, Z    +0.000, E1   +21.704, E3 +497796.618}
SPL {X  -162.820, Y  +491.396, Z    +0.000, E1   +21.707, E3 +497808.742}
SPL {X  -162.820, Y  +489.485, Z    +0.000, E1   +21.661, E3 +497819.089}
SPL {X  -162.820, Y  +487.723, Z    +0.000, E1   +21.665, E3 +497828.293}
SPL {X  -162.820, Y  +485.661, Z    +0.000, E1   +21.712, E3 +497838.736}
SPL {X  -162.820, Y  +482.775, Z    +0.000, E1   +21.716, E3 +497853.989}
SPL {X  -162.820, Y  +479.894, Z    +0.000, E1   +21.695, E3 +497869.065}
SPL {X  -162.820, Y  +477.685, Z    +0.000, E1   +21.656, E3 +497881.002}
SPL {X  -162.820, Y  +475.419, Z    +0.000, E1   +21.711, E3 +497892.355}
SPL {X  -162.820, Y  +473.301, Z    +0.000, E1   +21.712, E3 +497903.452}
SPL {X  -162.820, Y  +470.965, Z    +0.000, E1   +21.700, E3 +497915.797}
SPL {X  -162.820, Y  +469.036, Z    +0.000, E1   +21.695, E3 +497925.841}
SPL {X  -162.820, Y  +467.138, Z    +0.000, E1   +21.678, E3 +497936.012}
SPL {X  -162.820, Y  +465.011, Z    +0.000, E1   +21.692, E3 +497946.995}
SPL {X  -162.820, Y  +462.669, Z    +0.000, E1   +21.752, E3 +497958.776}
SPL {X  -162.820, Y  +460.725, Z    +0.000, E1   +21.689, E3 +497969.389}
SPL {X  -162.820, Y  +458.666, Z    +0.000, E1   +21.695, E3 +497980.201}
SPL {X  -162.820, Y  +456.431, Z    +0.000, E1   +21.708, E3 +497991.729}
SPL {X  -162.820, Y  +453.609, Z    +0.000, E1   +21.757, E3 +498006.263}
SPL {X  -162.820, Y  +450.610, Z    +0.000, E1   +21.698, E3 +498022.320}
SPL {X  -162.820, Y  +448.170, Z    +0.000, E1   +21.667, E3 +498035.341}
SPL {X  -162.820, Y  +446.246, Z    +0.000, E1   +21.696, E3 +498045.159}
SPL {X  -162.820, Y  +443.784, Z    +0.000, E1   +21.713, E3 +498057.945}
SPL {X  -162.820, Y  +440.567, Z    +0.000, E1   +21.731, E3 +498074.785}
SPL {X  -162.820, Y  +437.628, Z    +0.000, E1   +21.678, E3 +498090.449}
SPL {X  -162.820, Y  +435.262, Z    +0.000, E1   +21.727, E3 +498102.385}
SPL {X  -162.820, Y  +433.510, Z    +0.000, E1   +21.692, E3 +498111.798}
SPL {X  -162.820, Y  +431.492, Z    +0.000, E1   +21.686, E3 +498122.494}
SPL {X  -162.820, Y  +429.074, Z    +0.000, E1   +21.710, E3 +498134.946}
SPL {X  -162.820, Y  +427.020, Z    +0.000, E1   +21.674, E3 +498145.947}
SPL {X  -162.820, Y  +424.525, Z    +0.000, E1   +21.712, E3 +498158.860}
SPL {X  -162.820, Y  +421.144, Z    +0.000, E1   +21.719, E3 +498176.527}
SPL {X  -162.820, Y  +418.116, Z    +0.000, E1   +21.761, E3 +498191.858}
SPL {X  -162.820, Y  +416.127, Z    +0.000, E1   +21.715, E3 +498202.564}
SPL {X  -162.820, Y  +414.361, Z    +0.000, E1   +21.613, E3 +498212.751}
SPL {X  -162.820, Y  +412.134, Z    +0.000, E1   +21.697, E3 +498223.695}
SPL {X  -162.820, Y  +409.248, Z    +0.000, E1   +21.741, E3 +498238.631}
SPL {X  -162.820, Y  +406.238, Z    +0.000, E1   +21.697, E3 +498254.599}
SPL {X  -162.820, Y  +403.166, Z    +0.000, E1   +21.746, E3 +498270.405}
SPL {X  -162.820, Y  +400.348, Z    +0.000, E1   +21.713, E3 +498285.239}
SPL {X  -162.820, Y  +398.298, Z    +0.000, E1   +21.721, E3 +498295.855}
SPL {X  -162.820, Y  +396.371, Z    +0.000, E1   +21.713, E3 +498306.037}
SPL {X  -162.820, Y  +394.508, Z    +0.000, E1   +21.616, E3 +498316.592}
SPL {X  -162.820, Y  +391.777, Z    +0.000, E1   +21.714, E3 +498330.252}
SPL {X  -162.820, Y  +388.822, Z    +0.000, E1   +21.717, E3 +498345.571}
SPL {X  -162.820, Y  +386.818, Z    +0.000, E1   +21.679, E3 +498356.311}
SPL {X  -162.820, Y  +384.697, Z    +0.000, E1   +21.693, E3 +498367.381}
SPL {X  -162.820, Y  +382.288, Z    +0.000, E1   +21.742, E3 +498379.505}
SPL {X  -162.817, Y  +379.520, Z    +0.000, E1   +21.723, E3 +498394.343}
SPL {X  -162.776, Y  +376.710, Z    +0.000, E1   +21.698, E3 +498409.082}
SPL {X  -162.707, Y  +374.438, Z    +0.000, E1   +21.688, E3 +498421.085}
SPL {X  -162.607, Y  +372.171, Z    +0.000, E1   +21.692, E3 +498432.885}
SPL {X  -162.494, Y  +370.197, Z    +0.000, E1   +21.655, E3 +498443.511}
SPL {X  -162.349, Y  +368.131, Z    +0.000, E1   +21.624, E3 +498454.629}
SPL {X  -162.161, Y  +365.866, Z    +0.000, E1   +21.642, E3 +498466.315}
SPL {X  -161.651, Y  +361.024, Z    +0.000, E1   +22.970, E3 +498479.738}
SPL {X  -160.281, Y  +351.857, Z    +0.000, E1   +24.243, E3 +498515.077}
ENDSPLINE

SPLINE
SPL {X  -161.833, Y  +362.603, Z    +0.000, E1   +17.021, E3 +498529.773}
ENDSPLINE

SPLINE
SPL {X  -160.786, Y  +354.842, Z    +0.000, E1   +19.274, E3 +498561.928}
ENDSPLINE

SPLINE
SPL {X  -162.485, Y  +370.062, Z    +0.000, E1   +10.606, E3 +498568.307}
SPL {X  -162.818, Y  +379.636, Z    +0.000, E1    +5.115, E3 +498557.655}
SPL {X  -162.820, Y  +386.976, Z    +0.000, E1    +0.144, E3 +498556.755}
SPL {X  -162.820, Y  +390.236, Z    +0.000, E1    -2.204, E3 +498562.813}
SPL {X  -162.820, Y  +393.415, Z    +0.000, E1    -4.587, E3 +498564.097}
SPL {X  -162.820, Y  +399.630, Z    +0.000, E1    -9.426, E3 +498566.027}
SPL {X  -162.820, Y  +408.127, Z    +0.000, E1   -18.417, E3 +498552.315}
SPL {X  -162.820, Y  +420.083, Z    +0.000, E1   -24.325, E3 +498572.791}
SPL {X  -162.820, Y  +428.527, Z    +0.000, E1   -26.988, E3 +498590.083}
SPL {X  -162.820, Y  +431.336, Z    +0.000, E1   -24.162, E3 +498620.293}
SPL {X  -162.820, Y  +432.048, Z    +0.000, E1   -22.832, E3 +498634.797}
SPL {X  -162.820, Y  +434.888, Z    +0.000, E1   -22.823, E3 +498648.746}
SPL {X  -162.820, Y  +436.834, Z    +0.000, E1   -22.779, E3 +498658.706}
SPL {X  -162.820, Y  +438.868, Z    +0.000, E1   -22.837, E3 +498668.360}
SPL {X  -162.820, Y  +441.351, Z    +0.000, E1   -22.805, E3 +498680.935}
SPL {X  -162.820, Y  +443.809, Z    +0.000, E1   -22.804, E3 +498693.101}
SPL {X  -162.820, Y  +447.077, Z    +0.000, E1   -22.869, E3 +498708.912}
SPL {X  -162.820, Y  +449.911, Z    +0.000, E1   -22.774, E3 +498723.521}
SPL {X  -162.820, Y  +451.861, Z    +0.000, E1   -22.750, E3 +498733.369}
SPL {X  -162.820, Y  +454.167, Z    +0.000, E1   -22.842, E3 +498744.098}
SPL {X  -162.820, Y  +456.529, Z    +0.000, E1   -22.855, E3 +498755.627}
SPL {X  -162.820, Y  +458.725, Z    +0.000, E1   -22.793, E3 +498767.031}
SPL {X  -162.820, Y  +460.754, Z    +0.000, E1   -22.806, E3 +498776.904}
SPL {X  -162.820, Y  +462.409, Z    +0.000, E1   -22.783, E3 +498785.321}
SPL {X  -162.820, Y  +464.633, Z    +0.000, E1   -22.813, E3 +498796.150}
SPL {X  -162.820, Y  +467.913, Z    +0.000, E1   -22.879, E3 +498811.989}
SPL {X  -162.820, Y  +470.892, Z    +0.000, E1   -22.837, E3 +498826.879}
SPL {X  -162.820, Y  +472.726, Z    +0.000, E1   -22.777, E3 +498836.417}
SPL {X  -162.820, Y  +475.118, Z    +0.000, E1   -22.777, E3 +498848.389}
SPL {X  -162.820, Y  +478.177, Z    +0.000, E1   -22.834, E3 +498863.082}
SPL {X  -162.820, Y  +481.034, Z    +0.000, E1   -22.831, E3 +498877.219}
SPL {X  -162.820, Y  +483.391, Z    +0.000, E1   -22.793, E3 +498889.155}
SPL {X  -162.820, Y  +486.307, Z    +0.000, E1   -22.833, E3 +498903.409}
SPL {X  -162.820, Y  +489.750, Z    +0.000, E1   -22.832, E3 +498920.479}
SPL {X  -162.820, Y  +493.233, Z    +0.000, E1   -22.844, E3 +498937.616}
SPL {X  -162.820, Y  +496.150, Z    +0.000, E1   -22.796, E3 +498952.336}
SPL {X  -162.820, Y  +498.661, Z    +0.000, E1   -22.828, E3 +498964.516}
SPL {X  -162.820, Y  +501.761, Z    +0.000, E1   -22.820, E3 +498980.085}
SPL {X  -162.820, Y  +504.194, Z    +0.000, E1   -22.775, E3 +498992.276}
SPL {X  -162.820, Y  +506.908, Z    +0.000, E1   -22.877, E3 +499005.121}
SPL {X  -162.820, Y  +510.068, Z    +0.000, E1   -22.761, E3 +499021.592}
SPL {X  -162.820, Y  +512.359, Z    +0.000, E1   -22.823, E3 +499032.324}
SPL {X  -162.820, Y  +514.562, Z    +0.000, E1   -22.806, E3 +499043.510}
SPL {X  -162.820, Y  +517.952, Z    +0.000, E1   -22.864, E3 +499059.908}
SPL {X  -162.820, Y  +520.641, Z    +0.000, E1   -22.790, E3 +499073.626}
SPL {X  -162.820, Y  +522.740, Z    +0.000, E1   -22.811, E3 +499083.869}
SPL {X  -162.820, Y  +524.628, Z    +0.000, E1   -22.846, E3 +499092.864}
SPL {X  -162.820, Y  +526.661, Z    +0.000, E1   -22.801, E3 +499103.419}
SPL {X  -162.820, Y  +529.662, Z    +0.000, E1   -22.810, E3 +499118.270}
SPL {X  -162.820, Y  +532.614, Z    +0.000, E1   -22.828, E3 +499132.676}
SPL {X  -162.820, Y  +534.838, Z    +0.000, E1   -22.864, E3 +499143.305}
SPL {X  -162.820, Y  +536.882, Z    +0.000, E1   -22.782, E3 +499154.160}
SPL {X  -162.820, Y  +539.194, Z    +0.000, E1   -22.826, E3 +499165.208}
SPL {X  -162.820, Y  +541.555, Z    +0.000, E1   -22.817, E3 +499177.023}
SPL {X  -162.820, Y  +543.728, Z    +0.000, E1   -22.799, E3 +499187.880}
SPL {X  -162.820, Y  +545.925, Z    +0.000, E1   -22.803, E3 +499198.750}
SPL {X  -162.820, Y  +549.071, Z    +0.000, E1   -22.836, E3 +499214.278}
SPL {X  -162.820, Y  +553.089, Z    +0.000, E1   -22.838, E3 +499234.178}
SPL {X  -162.820, Y  +556.430, Z    +0.000, E1   -22.821, E3 +499250.679}
SPL {X  -162.820, Y  +559.675, Z    +0.000, E1   -22.837, E3 +499266.759}
SPL {X  -162.820, Y  +562.799, Z    +0.000, E1   -22.814, E3 +499282.265}
SPL {X  -162.820, Y  +565.170, Z    +0.000, E1   -22.801, E3 +499294.090}
SPL {X  -162.820, Y  +568.020, Z    +0.000, E1   -22.787, E3 +499308.477}
SPL {X  -162.820, Y  +570.992, Z    +0.000, E1   -22.834, E3 +499322.696}
SPL {X  -162.820, Y  +572.901, Z    +0.000, E1   -22.775, E3 +499332.564}
SPL {X  -162.820, Y  +575.638, Z    +0.000, E1   -22.855, E3 +499345.674}
SPL {X  -162.820, Y  +578.553, Z    +0.000, E1   -22.801, E3 +499360.386}
SPL {X  -162.820, Y  +581.064, Z    +0.000, E1   -22.823, E3 +499372.671}
SPL {X  -162.820, Y  +583.435, Z    +0.000, E1   -22.808, E3 +499384.492}
SPL {X  -162.820, Y  +585.410, Z    +0.000, E1   -22.764, E3 +499394.628}
SPL {X  -162.820, Y  +587.676, Z    +0.000, E1   -22.853, E3 +499405.143}
SPL {X  -162.820, Y  +590.707, Z    +0.000, E1   -22.855, E3 +499420.293}
SPL {X  -162.820, Y  +593.650, Z    +0.000, E1   -22.810, E3 +499435.053}
SPL {X  -162.820, Y  +595.830, Z    +0.000, E1   -22.828, E3 +499445.669}
SPL {X  -162.820, Y  +598.094, Z    +0.000, E1   -22.843, E3 +499456.782}
SPL {X  -162.820, Y  +600.420, Z    +0.000, E1   -22.826, E3 +499468.413}
SPL {X  -162.820, Y  +602.573, Z    +0.000, E1   -22.830, E3 +499478.999}
SPL {X  -162.820, Y  +604.828, Z    +0.000, E1   -22.784, E3 +499490.637}
SPL {X  -162.820, Y  +607.142, Z    +0.000, E1   -22.808, E3 +499501.818}
SPL {X  -162.820, Y  +608.890, Z    +0.000, E1   -22.790, E3 +499510.642}
SPL {X  -162.820, Y  +611.103, Z    +0.000, E1   -22.785, E3 +499521.680}
SPL {X  -162.820, Y  +613.294, Z    +0.000, E1   -22.780, E3 +499532.554}
SPL {X  -162.820, Y  +615.356, Z    +0.000, E1   -22.799, E3 +499542.611}
SPL {X  -162.820, Y  +617.439, Z    +0.000, E1   -22.808, E3 +499552.869}
SPL {X  -162.820, Y  +619.665, Z    +0.000, E1   -22.817, E3 +499563.837}
SPL {X  -162.820, Y  +621.733, Z    +0.000, E1   -22.759, E3 +499574.561}
SPL {X  -162.820, Y  +624.076, Z    +0.000, E1   -22.774, E3 +499586.066}
SPL {X  -162.820, Y  +626.527, Z    +0.000, E1   -22.768, E3 +499598.309}
SPL {X  -162.820, Y  +629.758, Z    +0.000, E1   -22.800, E3 +499614.238}
SPL {X  -162.820, Y  +632.572, Z    +0.000, E1   -22.785, E3 +499628.087}
SPL {X  -162.820, Y  +634.507, Z    +0.000, E1   -22.784, E3 +499637.726}
SPL {X  -162.820, Y  +636.863, Z    +0.000, E1   -22.760, E3 +499649.648}
SPL {X  -162.820, Y  +640.111, Z    +0.000, E1   -22.809, E3 +499665.531}
SPL {X  -162.820, Y  +643.449, Z    +0.000, E1   -22.796, E3 +499682.049}
SPL {X  -162.820, Y  +645.630, Z    +0.000, E1   -22.795, E3 +499692.745}
SPL {X  -162.820, Y  +647.561, Z    +0.000, E1   -22.705, E3 +499703.195}
SPL {X  -162.820, Y  +649.758, Z    +0.000, E1   -22.780, E3 +499713.385}
SPL {X  -162.820, Y  +651.708, Z    +0.000, E1   -22.810, E3 +499722.880}
SPL {X  -162.820, Y  +653.898, Z    +0.000, E1   -22.796, E3 +499733.801}
SPL {X  -162.820, Y  +656.161, Z    +0.000, E1   -22.812, E3 +499744.922}
SPL {X  -162.820, Y  +658.384, Z    +0.000, E1   -22.822, E3 +499755.788}
SPL {X  -162.820, Y  +660.215, Z    +0.000, E1   -22.649, E3 +499766.379}
SPL {X  -162.820, Y  +662.823, Z    +0.000, E1   -22.799, E3 +499778.087}
SPL {X  -162.820, Y  +665.862, Z    +0.000, E1   -22.864, E3 +499792.786}
SPL {X  -162.820, Y  +668.960, Z    +0.000, E1   -22.773, E3 +499808.737}
SPL {X  -162.820, Y  +671.605, Z    +0.000, E1   -22.777, E3 +499821.811}
SPL {X  -162.817, Y  +674.515, Z    +0.000, E1   -22.816, E3 +499836.008}
SPL {X  -162.773, Y  +677.428, Z    +0.000, E1   -22.762, E3 +499850.816}
SPL {X  -162.691, Y  +679.987, Z    +0.000, E1   -22.794, E3 +499863.229}
SPL {X  -162.604, Y  +681.880, Z    +0.000, E1   -22.691, E3 +499873.390}
SPL {X  -162.458, Y  +684.346, Z    +0.000, E1   -22.764, E3 +499885.184}
SPL {X  -162.296, Y  +686.547, Z    +0.000, E1   -22.660, E3 +499896.800}
SPL {X  -162.164, Y  +688.106, Z    +0.000, E1   -22.661, E3 +499904.534}
SPL {X  -161.938, Y  +690.422, Z    +0.000, E1   -22.769, E3 +499915.209}
SPL {X  -161.065, Y  +697.344, Z    +0.000, E1   -25.698, E3 +499924.329}
SPL {X  -158.553, Y  +710.529, Z    +0.000, E1   -30.890, E3 +499938.226}
ENDSPLINE

SPLINE
SPL {X  -161.215, Y  +696.305, Z    +0.000, E1   -20.575, E3 +499964.806}
SPL {X  -161.691, Y  +692.643, Z    +0.000, E1   -17.369, E3 +499980.994}
SPL {X  -162.534, Y  +683.153, Z    +0.000, E1   -10.475, E3 +500006.462}
SPL {X  -162.820, Y  +670.105, Z    +0.000, E1    -2.484, E3 +499999.108}
SPL {X  -162.820, Y  +665.819, Z    +0.000, E1    +0.492, E3 +500001.405}
SPL {X  -162.820, Y  +661.883, Z    +0.000, E1    +3.373, E3 +500005.881}
SPL {X  -162.820, Y  +655.163, Z    +0.000, E1    +8.702, E3 +500005.480}
SPL {X  -162.820, Y  +634.515, Z    +0.000, E1   +26.439, E3 +499997.893}
ENDSPLINE

SPLINE
SPL {X  -162.820, Y  +638.080, Z    +0.000, E1   +18.858, E3 +500027.858}
ENDSPLINE

SPLINE
SPL {X  -162.820, Y  +623.278, Z    +0.000, E1   +28.723, E3 +500029.428}
SPL {X  -162.820, Y  +618.658, Z    +0.000, E1   +26.841, E3 +500058.037}
ENDSPLINE

SPLINE
SPL {X  -162.820, Y  +623.685, Z    +0.000, E1   +22.346, E3 +500070.344}
ENDSPLINE

SPLINE
SPL {X  -162.820, Y  +621.304, Z    +0.000, E1   +22.259, E3 +500083.159}
SPL {X  -162.820, Y  +618.758, Z    +0.000, E1   +22.239, E3 +500096.310}
SPL {X  -162.820, Y  +616.062, Z    +0.000, E1   +22.275, E3 +500109.730}
SPL {X  -162.820, Y  +613.536, Z    +0.000, E1   +22.242, E3 +500122.852}
SPL {X  -162.820, Y  +610.461, Z    +0.000, E1   +22.264, E3 +500138.483}
SPL {X  -162.820, Y  +607.796, Z    +0.000, E1   +22.261, E3 +500151.854}
SPL {X  -162.820, Y  +605.178, Z    +0.000, E1   +22.267, E3 +500165.338}
SPL {X  -162.820, Y  +602.350, Z    +0.000, E1   +22.224, E3 +500179.955}
SPL {X  -162.820, Y  +599.842, Z    +0.000, E1   +22.298, E3 +500192.107}
SPL {X  -162.820, Y  +597.194, Z    +0.000, E1   +22.253, E3 +500206.028}
SPL {X  -162.820, Y  +594.779, Z    +0.000, E1   +22.284, E3 +500217.932}
SPL {X  -162.820, Y  +592.389, Z    +0.000, E1   +22.245, E3 +500230.548}
SPL {X  -162.820, Y  +589.492, Z    +0.000, E1   +22.304, E3 +500244.733}
SPL {X  -162.820, Y  +587.447, Z    +0.000, E1   +22.279, E3 +500255.262}
SPL {X  -162.820, Y  +585.192, Z    +0.000, E1   +22.298, E3 +500266.672}
SPL {X  -162.820, Y  +582.610, Z    +0.000, E1   +22.234, E3 +500280.295}
SPL {X  -162.820, Y  +580.317, Z    +0.000, E1   +22.300, E3 +500291.349}
SPL {X  -162.820, Y  +578.878, Z    +0.000, E1   +22.272, E3 +500298.858}
SPL {X  -162.820, Y  +576.856, Z    +0.000, E1   +22.233, E3 +500309.617}
SPL {X  -162.820, Y  +574.811, Z    +0.000, E1   +22.236, E3 +500319.880}
SPL {X  -162.820, Y  +572.645, Z    +0.000, E1   +22.246, E3 +500330.976}
SPL {X  -162.820, Y  +570.282, Z    +0.000, E1   +22.231, E3 +500343.026}
SPL {X  -162.820, Y  +567.961, Z    +0.000, E1   +22.247, E3 +500354.816}
SPL {X  -162.820, Y  +564.506, Z    +0.000, E1   +22.298, E3 +500372.130}
SPL {X  -162.820, Y  +561.620, Z    +0.000, E1   +22.191, E3 +500387.511}
SPL {X  -162.820, Y  +559.515, Z    +0.000, E1   +22.273, E3 +500397.513}
SPL {X  -162.820, Y  +556.723, Z    +0.000, E1   +22.309, E3 +500411.596}
SPL {X  -162.820, Y  +554.378, Z    +0.000, E1   +22.288, E3 +500423.442}
SPL {X  -162.820, Y  +552.787, Z    +0.000, E1   +22.213, E3 +500432.264}
SPL {X  -162.820, Y  +550.871, Z    +0.000, E1   +22.229, E3 +500441.858}
SPL {X  -162.820, Y  +548.168, Z    +0.000, E1   +22.298, E3 +500455.194}
SPL {X  -162.820, Y  +545.860, Z    +0.000, E1   +22.216, E3 +500467.452}
SPL {X  -162.820, Y  +543.558, Z    +0.000, E1   +22.285, E3 +500478.682}
SPL {X  -162.820, Y  +541.633, Z    +0.000, E1   +22.257, E3 +500488.611}
SPL {X  -162.820, Y  +539.116, Z    +0.000, E1   +22.302, E3 +500501.221}
SPL {X  -162.820, Y  +535.523, Z    +0.000, E1   +22.266, E3 +500519.883}
SPL {X  -162.820, Y  +531.757, Z    +0.000, E1   +22.276, E3 +500538.937}
SPL {X  -162.820, Y  +527.980, Z    +0.000, E1   +22.326, E3 +500557.768}
SPL {X  -162.820, Y  +524.599, Z    +0.000, E1   +22.287, E3 +500575.166}
SPL {X  -162.820, Y  +522.011, Z    +0.000, E1   +22.282, E3 +500588.243}
SPL {X  -162.820, Y  +519.457, Z    +0.000, E1   +22.481, E3 +500599.532}
SPL {X  -162.820, Y  +506.285, Z    +0.000, E1   +28.538, E3 +500610.990}
SPL {X  -162.820, Y  +504.441, Z    +0.000, E1   +27.574, E3 +500625.332}
SPL {X  -162.820, Y  +502.813, Z    +0.000, E1   +26.013, E3 +500643.530}
SPL {X  -162.820, Y  +502.016, Z    +0.000, E1   +24.802, E3 +500655.873}
SPL {X  -162.820, Y  +501.060, Z    +0.000, E1   +24.081, E3 +500666.062}
SPL {X  -162.820, Y  +500.336, Z    +0.000, E1   +23.110, E3 +500677.202}
SPL {X  -162.820, Y  +499.240, Z    +0.000, E1   +22.316, E3 +500689.513}
SPL {X  -162.820, Y  +498.027, Z    +0.000, E1   +21.516, E3 +500702.420}
SPL {X  -162.820, Y  +495.897, Z    +0.000, E1   +21.662, E3 +500712.341}
SPL {X  -162.820, Y  +493.717, Z    +0.000, E1   +21.704, E3 +500723.447}
SPL {X  -162.820, Y  +491.396, Z    +0.000, E1   +21.707, E3 +500735.571}
SPL {X  -162.820, Y  +488.560, Z    +0.000, E1   +21.695, E3 +500750.680}
SPL {X  -162.820, Y  +485.661, Z    +0.000, E1   +21.712, E3 +500765.566}
SPL {X  -162.820, Y  +483.668, Z    +0.000, E1   +21.664, E3 +500776.393}
SPL {X  -162.820, Y  +481.739, Z    +0.000, E1   +21.704, E3 +500786.107}
SPL {X  -162.820, Y  +479.894, Z    +0.000, E1   +21.695, E3 +500795.894}
SPL {X  -162.820, Y  +477.685, Z    +0.000, E1   +21.656, E3 +500807.832}
SPL {X  -162.820, Y  +475.419, Z    +0.000, E1   +21.711, E3 +500819.184}
SPL {X  -162.820, Y  +473.301, Z    +0.000, E1   +21.712, E3 +500830.282}
SPL {X  -162.820, Y  +470.965, Z    +0.000, E1   +21.700, E3 +500842.626}
SPL {X  -162.820, Y  +469.036, Z    +0.000, E1   +21.695, E3 +500852.670}
SPL {X  -162.820, Y  +467.138, Z    +0.000, E1   +21.678, E3 +500862.842}
SPL {X  -162.820, Y  +465.011, Z    +0.000, E1   +21.692, E3 +500873.824}
SPL {X  -162.820, Y  +462.669, Z    +0.000, E1   +21.752, E3 +500885.605}
SPL {X  -162.820, Y  +460.725, Z    +0.000, E1   +21.689, E3 +500896.218}
SPL {X  -162.820, Y  +458.666, Z    +0.000, E1   +21.695, E3 +500907.030}
SPL {X  -162.820, Y  +456.431, Z    +0.000, E1   +21.708, E3 +500918.558}
SPL {X  -162.820, Y  +453.609, Z    +0.000, E1   +21.757, E3 +500933.092}
SPL {X  -162.820, Y  +450.610, Z    +0.000, E1   +21.698, E3 +500949.150}
SPL {X  -162.820, Y  +448.170, Z    +0.000, E1   +21.667, E3 +500962.170}
SPL {X  -162.820, Y  +446.246, Z    +0.000, E1   +21.696, E3 +500971.988}
SPL {X  -162.820, Y  +443.784, Z    +0.000, E1   +21.713, E3 +500984.774}
SPL {X  -162.820, Y  +440.567, Z    +0.000, E1   +21.731, E3 +501001.614}
SPL {X  -162.820, Y  +437.628, Z    +0.000, E1   +21.678, E3 +501017.278}
SPL {X  -162.820, Y  +434.473, Z    +0.000, E1   +21.747, E3 +501033.374}
SPL {X  -162.820, Y  +431.492, Z    +0.000, E1   +21.686, E3 +501049.323}
SPL {X  -162.820, Y  +429.074, Z    +0.000, E1   +21.710, E3 +501061.775}
SPL {X  -162.820, Y  +426.023, Z    +0.000, E1   +21.718, E3 +501077.843}
SPL {X  -162.820, Y  +422.986, Z    +0.000, E1   +21.685, E3 +501093.890}
SPL {X  -162.820, Y  +420.528, Z    +0.000, E1   +21.706, E3 +501106.540}
SPL {X  -162.820, Y  +418.116, Z    +0.000, E1   +21.761, E3 +501118.688}
SPL {X  -162.820, Y  +416.127, Z    +0.000, E1   +21.715, E3 +501129.393}
SPL {X  -162.820, Y  +414.361, Z    +0.000, E1   +21.613, E3 +501139.580}
SPL {X  -162.820, Y  +412.134, Z    +0.000, E1   +21.697, E3 +501150.525}
SPL {X  -162.820, Y  +409.248, Z    +0.000, E1   +21.741, E3 +501165.460}
SPL {X  -162.820, Y  +406.238, Z    +0.000, E1   +21.697, E3 +501181.428}
SPL {X  -162.820, Y  +404.001, Z    +0.000, E1   +21.723, E3 +501192.858}
SPL {X  -162.820, Y  +402.223, Z    +0.000, E1   +21.697, E3 +501202.343}
SPL {X  -162.820, Y  +400.348, Z    +0.000, E1   +21.713, E3 +501212.069}
SPL {X  -162.820, Y  +398.298, Z    +0.000, E1   +21.721, E3 +501222.684}
SPL {X  -162.820, Y  +396.371, Z    +0.000, E1   +21.713, E3 +501232.866}
SPL {X  -162.820, Y  +394.508, Z    +0.000, E1   +21.616, E3 +501243.422}
SPL {X  -162.820, Y  +392.435, Z    +0.000, E1   +21.681, E3 +501253.775}
SPL {X  -162.820, Y  +389.390, Z    +0.000, E1   +21.742, E3 +501269.382}
SPL {X  -162.820, Y  +386.818, Z    +0.000, E1   +21.679, E3 +501283.140}
SPL {X  -162.820, Y  +384.697, Z    +0.000, E1   +21.693, E3 +501294.211}
SPL {X  -162.820, Y  +382.288, Z    +0.000, E1   +21.742, E3 +501306.334}
SPL {X  -162.820, Y  +380.381, Z    +0.000, E1   +21.655, E3 +501317.059}
SPL {X  -162.808, Y  +378.512, Z    +0.000, E1   +21.736, E3 +501326.112}
SPL {X  -162.776, Y  +376.710, Z    +0.000, E1   +21.698, E3 +501335.911}
SPL {X  -162.707, Y  +374.438, Z    +0.000, E1   +21.688, E3 +501347.915}
SPL {X  -162.607, Y  +372.171, Z    +0.000, E1   +21.692, E3 +501359.714}
SPL {X  -162.494, Y  +370.197, Z    +0.000, E1   +21.655, E3 +501370.341}
SPL {X  -162.349, Y  +368.131, Z    +0.000, E1   +21.624, E3 +501381.459}
SPL {X  -162.161, Y  +365.866, Z    +0.000, E1   +21.642, E3 +501393.144}
SPL {X  -161.927, Y  +363.466, Z    +0.000, E1   +21.730, E3 +501404.915}
SPL {X  -160.290, Y  +351.907, Z    +0.000, E1   +27.562, E3 +501412.493}
SPL {X  -159.725, Y  +348.905, Z    +0.000, E1   +26.136, E3 +501437.728}
ENDSPLINE

SPLINE
SPL {X  -160.871, Y  +355.385, Z    +0.000, E1   +21.841, E3 +501446.571}
SPL {X  -161.833, Y  +362.603, Z    +0.000, E1   +17.021, E3 +501456.602}
ENDSPLINE

SPLINE
SPL {X  -160.786, Y  +354.842, Z    +0.000, E1   +19.274, E3 +501488.758}
ENDSPLINE

